KUKA KRL program: EPS_2_251825_SA30_A_20260116064111.src

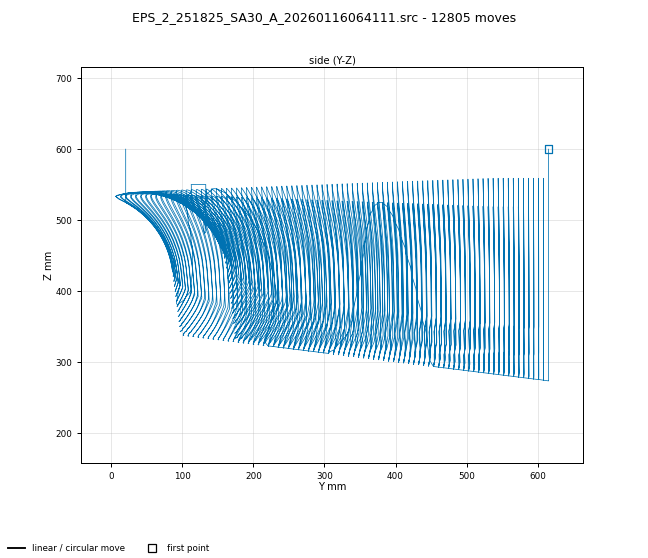
[picture p0: tool path of EPS_2_251825_SA30_A_20260116064111.src, 12805 of 12807 moves have a stored position in this frame; points joined in program order, loops and branches not executed]
&ACCESS RVP
&REL 4
&COMMENT QRS 19112012
&PARAM EDITMASK = *
DEF PART()
EXT BAS (BAS_COMMAND :IN,REAL :IN )
INT I
BAS (#INITMOV,0 )

;KUKA QRS Post kuka4.cps  Date:22-06-2017 !

File_ID=2989

QRS_PRE_INIT()

;Init var - Until changes are made in qrs_pre_init
Outlet_Square_prg=0
Inlet_1_Square_prg=0
Inlet_2_Square_prg=0
Inlet_3_Square_prg=0
Inlet_4_Square_prg=0
Inlet_5_Square_prg=0

Outlet_1={X 0.000, Y 535.490, Z 458.500, B 0.000, E1 0.000 }
Inlet_1={X 0.000, Y 538.340, Z 418.500, B 0.000, E1 194.000 }
Outlet_1_type=201
Inlet_1_type=201
;QRS#1=Sidecore dimensions
;QRS#2=200-8" PVC SDR 35
;QRS#3=200-8" PVC SDR 35
;QRS#4=
;QRS#5=
;QRS#6=
;QRS#7=
;QRS#8=
;QRS#9=12-08 PSX
;QRS#10=12-08 PSX
;QRS#11=
;QRS#12=
;QRS#13=
;QRS#14=
;QRS#15=
;QRS#16=1220x127x838 2,75'
;QRS#17=EPS Height
;QRS#18=559
;QRS#19=*
;QRS#20= UPDATED VERSION 22-06-2017
;QRS#21=*
Outlet_Square=0100
Inlet_1_Square=0100
Inlet_2_Square=0
Inlet_3_Square=0
Inlet_4_Square=0
Inlet_5_Square=0
Mill_Square=1
Outlet_Square_Prg=204
Inlet_1_Square_prg=204

QRS_INIT()

$ADVANCE=5

; T1
PTP {E1 173.624,E2 173.624}
PTP {X 0,Y 615.46,A -85,B 0,C 180,E1 173.624,E2 173.624,E3 0,E4 0,E5 0,E6 0}
QRS_SPEED_INIT()
LIN {X 0,Y 615.46,Z 600,A -85,B 0,C 180,E1 173.624,E2 173.624,E3 0,E4 0,E5 0,E6 0} C_VEL
LIN {X 0,Y 615.46,Z 283.872,A -85,B 0,C 180,E1 173.624,E2 173.624} C_VEL
LIN {X 0,Y 615.46,Z 275.69,A -85,B 0,C 180,E1 173.624,E2 173.624} C_VEL
LIN {X 0,Y 615.454,Z 273.69,A -85,B 0,C 180,E1 173.438,E2 173.438} C_VEL
LIN {X 0,Y 615.487,Z 273.682,A -85,B 0,C 180,E1 170.801,E2 170.801} C_VEL
LIN {X 0,Y 615.494,Z 273.696,A -85,B 0,C 180,E1 168.139,E2 168.139} C_VEL
LIN {X 0,Y 615.455,Z 273.694,A -85,B 0,C 180,E1 165.45,E2 165.45} C_VEL
LIN {X 0,Y 615.454,Z 273.694,A -85,B 0,C 180,E1 163.412,E2 163.412} C_VEL
LIN {X 0,Y 615.454,Z 273.694,A -85,B 0,C 180,E1 161.353,E2 161.353} C_VEL
LIN {X 0,Y 615.452,Z 273.694,A -85,B 0,C 180,E1 159.268,E2 159.268} C_VEL
LIN {X 0,Y 615.449,Z 273.694,A -85,B 0,C 180,E1 157.154,E2 157.154} C_VEL
LIN {X 0,Y 615.446,Z 273.693,A -85,B 0,C 180,E1 155.006,E2 155.006} C_VEL
LIN {X 0,Y 615.444,Z 273.692,A -85,B 0,C 180,E1 152.821,E2 152.821} C_VEL
LIN {X 0,Y 615.474,Z 273.686,A -85,B 0,C 180,E1 150.205,E2 150.205} C_VEL
LIN {X 0,Y 615.493,Z 273.698,A -85,B 0,C 180,E1 147.543,E2 147.543} C_VEL
LIN {X 0,Y 615.47,Z 273.698,A -85,B 0,C 180,E1 145.184,E2 145.184} C_VEL
LIN {X 0,Y 615.443,Z 273.695,A -85,B 0,C 180,E1 142.754,E2 142.754} C_VEL
LIN {X 0,Y 615.465,Z 273.688,A -85,B 0,C 180,E1 139.912,E2 139.912} C_VEL
LIN {X 0,Y 615.466,Z 273.699,A -85,B 0,C 180,E1 136.953,E2 136.953} C_VEL
LIN {X 0,Y 615.473,Z 273.698,A -85,B 0,C 180,E1 134.93,E2 134.93} C_VEL
LIN {X 0,Y 615.435,Z 273.695,A -85,B 0,C 180,E1 132.356,E2 132.356} C_VEL
LIN {X 0,Y 615.433,Z 273.693,A -85,B 0,C 180,E1 130.083,E2 130.083} C_VEL
LIN {X 0,Y 615.432,Z 273.693,A -85,B 0,C 180,E1 128.005,E2 128.005} C_VEL
LIN {X 0,Y 615.446,Z 273.692,A -85,B 0,C 180,E1 125.617,E2 125.617} C_VEL
LIN {X 0,Y 615.473,Z 273.691,A -85,B 0,C 180,E1 123.236,E2 123.236} C_VEL
LIN {X 0,Y 615.492,Z 273.695,A -85,B 0,C 180,E1 120.918,E2 120.918} C_VEL
LIN {X 0,Y 615.426,Z 273.696,A -85,B 0,C 180,E1 117.917,E2 117.917} C_VEL
LIN {X 0,Y 615.427,Z 273.694,A -85,B 0,C 180,E1 115.556,E2 115.556} C_VEL
LIN {X 0,Y 615.484,Z 273.692,A -85,B 0,C 180,E1 112.844,E2 112.844} C_VEL
LIN {X 0,Y 615.442,Z 273.698,A -85,B 0,C 180,E1 110.034,E2 110.034} C_VEL
LIN {X 0,Y 615.44,Z 273.698,A -85,B 0,C 180,E1 107.958,E2 107.958} C_VEL
LIN {X 0,Y 615.439,Z 273.699,A -85,B 0,C 180,E1 105.906,E2 105.906} C_VEL
LIN {X 0,Y 615.441,Z 273.699,A -85,B 0,C 180,E1 103.875,E2 103.875} C_VEL
LIN {X 0,Y 615.445,Z 273.699,A -85,B 0,C 180,E1 101.861,E2 101.861} C_VEL
LIN {X 0,Y 615.45,Z 273.699,A -85,B 0,C 180,E1 99.862,E2 99.862} C_VEL
LIN {X 0,Y 615.411,Z 273.698,A -85,B 0,C 180,E1 97.216,E2 97.216} C_VEL
LIN {X 0,Y 615.43,Z 273.697,A -85,B 0,C 180,E1 94.666,E2 94.666} C_VEL
LIN {X 0,Y 615.473,Z 275.838,A -85,B 0,C 180,E1 94.256,E2 94.256} C_VEL
LIN {X 0,Y 615.449,Z 291.323,A -85,B 0,C 180,E1 91.635,E2 91.635} C_VEL
LIN {X 0,Y 615.455,Z 306.957,A -85,B 0,C 180,E1 89.018,E2 89.018} C_VEL
LIN {X 0,Y 615.468,Z 308.181,A -85,B 0,C 180,E1 88.814,E2 88.814} C_VEL
LIN {X 0,Y 615.469,Z 414.797,A -85,B 0,C 180,E1 87.545,E2 87.545} C_VEL
LIN {X 0,Y 615.464,Z 427.886,A -85,B 0,C 180,E1 87.259,E2 87.259} C_VEL
LIN {X 0,Y 615.484,Z 440.419,A -85,B 0,C 180,E1 86.849,E2 86.849} C_VEL
LIN {X 0,Y 615.484,Z 452.453,A -85,B 0,C 180,E1 86.317,E2 86.317} C_VEL
LIN {X 0,Y 615.494,Z 463.84,A -85,B 0,C 180,E1 85.661,E2 85.661} C_VEL
LIN {X 0,Y 615.498,Z 474.118,A -85,B 0,C 180,E1 84.923,E2 84.923} C_VEL
LIN {X 0,Y 615.497,Z 481.621,A -85,B 0,C 180,E1 84.266,E2 84.266} C_VEL
LIN {X 0,Y 615.496,Z 489.878,A -85,B 0,C 180,E1 83.417,E2 83.417} C_VEL
LIN {X 0,Y 615.49,Z 497.479,A -85,B 0,C 180,E1 82.454,E2 82.454} C_VEL
LIN {X 0,Y 615.496,Z 503.742,A -85,B 0,C 180,E1 81.463,E2 81.463} C_VEL
LIN {X 0,Y 615.497,Z 508.742,A -85,B 0,C 180,E1 80.469,E2 80.469} C_VEL
LIN {X 0,Y 615.496,Z 512.615,A -85,B 0,C 180,E1 79.473,E2 79.473} C_VEL
LIN {X 0,Y 615.497,Z 514.607,A -85,B 0,C 180,E1 78.807,E2 78.807} C_VEL
LIN {X 0,Y 615.495,Z 516.186,A -85,B 0,C 180,E1 78.139,E2 78.139} C_VEL
LIN {X 0,Y 615.495,Z 517.337,A -85,B 0,C 180,E1 77.47,E2 77.47} C_VEL
LIN {X 0,Y 615.495,Z 518.354,A -85,B 0,C 180,E1 76.126,E2 76.126} C_VEL
LIN {X 0,Y 615.497,Z 518.271,A -85,B 0,C 180,E1 75.451,E2 75.451} C_VEL
LIN {X 0,Y 615.494,Z 517.731,A -85,B 0,C 180,E1 74.774,E2 74.774} C_VEL
LIN {X 0,Y 615.493,Z 515.746,A -85,B 0,C 180,E1 73.568,E2 73.568} C_VEL
LIN {X 0,Y 615.496,Z 512.453,A -85,B 0,C 180,E1 72.387,E2 72.387} C_VEL
LIN {X 0,Y 615.497,Z 508.371,A -85,B 0,C 180,E1 71.354,E2 71.354} C_VEL
LIN {X 0,Y 615.497,Z 501.94,A -85,B 0,C 180,E1 70.141,E2 70.141} C_VEL
LIN {X 0,Y 615.498,Z 494.801,A -85,B 0,C 180,E1 69.094,E2 69.094} C_VEL
LIN {X 0,Y 615.499,Z 487.402,A -85,B 0,C 180,E1 68.216,E2 68.216} C_VEL
LIN {X 0,Y 615.496,Z 477.643,A -85,B 0,C 180,E1 67.28,E2 67.28} C_VEL
LIN {X 0,Y 615.483,Z 466.81,A -85,B 0,C 180,E1 66.443,E2 66.443} C_VEL
LIN {X 0,Y 615.46,Z 456.253,A -85,B 0,C 180,E1 65.795,E2 65.795} C_VEL
LIN {X 0,Y 615.495,Z 444.674,A -85,B 0,C 180,E1 65.234,E2 65.234} C_VEL
LIN {X 0,Y 615.448,Z 431.759,A -85,B 0,C 180,E1 64.761,E2 64.761} C_VEL
LIN {X 0,Y 615.428,Z 419.153,A -85,B 0,C 180,E1 64.443,E2 64.443} C_VEL
LIN {X 0,Y 615.426,Z 403.17,A -85,B 0,C 180,E1 64.213,E2 64.213} C_VEL
LIN {X 0,Y 615.497,Z 308.127,A -85,B 0,C 180,E1 63.089,E2 63.089} C_VEL
LIN {X 0,Y 615.459,Z 292.076,A -85,B 0,C 180,E1 60.401,E2 60.401} C_VEL
LIN {X 0,Y 615.486,Z 275.929,A -85,B 0,C 180,E1 57.67,E2 57.67} C_VEL
LIN {X 0,Y 615.48,Z 273.686,A -85,B 0,C 180,E1 57.251,E2 57.251} C_VEL
LIN {X 0,Y 615.479,Z 273.686,A -85,B 0,C 180,E1 55.184,E2 55.184} C_VEL
LIN {X 0,Y 615.489,Z 273.68,A -85,B 0,C 180,E1 52.758,E2 52.758} C_VEL
LIN {X 0,Y 615.477,Z 273.694,A -85,B 0,C 180,E1 49.913,E2 49.913} C_VEL
LIN {X 0,Y 615.49,Z 273.698,A -85,B 0,C 180,E1 47.647,E2 47.647} C_VEL
LIN {X 0,Y 615.477,Z 273.688,A -85,B 0,C 180,E1 44.931,E2 44.931} C_VEL
LIN {X 0,Y 615.477,Z 273.685,A -85,B 0,C 180,E1 42.079,E2 42.079} C_VEL
LIN {X 0,Y 615.474,Z 273.69,A -85,B 0,C 180,E1 39.751,E2 39.751} C_VEL
LIN {X 0,Y 615.481,Z 273.694,A -85,B 0,C 180,E1 36.936,E2 36.936} C_VEL
LIN {X 0,Y 615.49,Z 273.68,A -85,B 0,C 180,E1 34.022,E2 34.022} C_VEL
LIN {X 0,Y 615.481,Z 273.702,A -85,B 0,C 180,E1 31.085,E2 31.085} C_VEL
LIN {X 0,Y 615.476,Z 273.689,A -85,B 0,C 180,E1 28.449,E2 28.449} C_VEL
LIN {X 0,Y 615.488,Z 273.681,A -85,B 0,C 180,E1 25.716,E2 25.716} C_VEL
LIN {X 0,Y 615.491,Z 273.699,A -85,B 0,C 180,E1 22.845,E2 22.845} C_VEL
LIN {X 0,Y 615.477,Z 273.686,A -85,B 0,C 180,E1 20.033,E2 20.033} C_VEL
LIN {X 0,Y 615.477,Z 273.685,A -85,B 0,C 180,E1 17.271,E2 17.271} C_VEL
LIN {X 0,Y 615.491,Z 273.7,A -85,B 0,C 180,E1 14.549,E2 14.549} C_VEL
LIN {X 0,Y 615.474,Z 273.688,A -85,B 0,C 180,E1 11.861,E2 11.861} C_VEL
LIN {X 0,Y 615.491,Z 273.68,A -85,B 0,C 180,E1 9.199,E2 9.199} C_VEL
LIN {X 0,Y 615.476,Z 273.694,A -85,B 0,C 180,E1 6.557,E2 6.557} C_VEL
LIN {X 0,Y 615.482,Z 273.695,A -85,B 0,C 180,E1 3.929,E2 3.929} C_VEL
LIN {X 0,Y 615.48,Z 273.683,A -85,B 0,C 180,E1 1.309,E2 1.309} C_VEL
LIN {X 0,Y 615.482,Z 273.684,A -85,B 0,C 180,E1 -1.309,E2 -1.309} C_VEL
LIN {X 0,Y 615.487,Z 273.696,A -85,B 0,C 180,E1 -3.928,E2 -3.928} C_VEL
LIN {X 0,Y 615.475,Z 273.692,A -85,B 0,C 180,E1 -6.57,E2 -6.57} C_VEL
LIN {X 0,Y 615.49,Z 273.68,A -85,B 0,C 180,E1 -9.199,E2 -9.199} C_VEL
LIN {X 0,Y 615.477,Z 273.689,A -85,B 0,C 180,E1 -11.861,E2 -11.861} C_VEL
LIN {X 0,Y 615.489,Z 273.698,A -85,B 0,C 180,E1 -14.549,E2 -14.549} C_VEL
LIN {X 0,Y 615.475,Z 273.685,A -85,B 0,C 180,E1 -17.271,E2 -17.271} C_VEL
LIN {X 0,Y 615.479,Z 273.686,A -85,B 0,C 180,E1 -20.033,E2 -20.033} C_VEL
LIN {X 0,Y 615.486,Z 273.697,A -85,B 0,C 180,E1 -22.845,E2 -22.845} C_VEL
LIN {X 0,Y 615.487,Z 273.681,A -85,B 0,C 180,E1 -25.716,E2 -25.716} C_VEL
LIN {X 0,Y 615.485,Z 273.695,A -85,B 0,C 180,E1 -28.658,E2 -28.658} C_VEL
LIN {X 0,Y 615.481,Z 273.699,A -85,B 0,C 180,E1 -31.085,E2 -31.085} C_VEL
LIN {X 0,Y 615.489,Z 273.68,A -85,B 0,C 180,E1 -34.022,E2 -34.022} C_VEL
LIN {X 0,Y 615.484,Z 273.695,A -85,B 0,C 180,E1 -36.936,E2 -36.936} C_VEL
LIN {X 0,Y 615.47,Z 273.689,A -85,B 0,C 180,E1 -39.752,E2 -39.752} C_VEL
LIN {X 0,Y 615.493,Z 273.679,A -85,B 0,C 180,E1 -42.353,E2 -42.353} C_VEL
LIN {X 0,Y 615.481,Z 273.692,A -85,B 0,C 180,E1 -45.069,E2 -45.069} C_VEL
LIN {X 0,Y 615.47,Z 273.692,A -85,B 0,C 180,E1 -47.922,E2 -47.922} C_VEL
LIN {X 0,Y 615.471,Z 273.686,A -85,B 0,C 180,E1 -50.249,E2 -50.249} C_VEL
LIN {X 0,Y 615.481,Z 273.686,A -85,B 0,C 180,E1 -53.065,E2 -53.065} C_VEL
LIN {X 0,Y 615.48,Z 273.696,A -85,B 0,C 180,E1 -55.978,E2 -55.978} C_VEL
LIN {X 0,Y 615.469,Z 273.69,A -85,B 0,C 180,E1 -58.313,E2 -58.313} C_VEL
LIN {X 0,Y 615.47,Z 273.686,A -85,B 0,C 180,E1 -60.593,E2 -60.593} C_VEL
LIN {X 0,Y 615.486,Z 273.681,A -85,B 0,C 180,E1 -62.956,E2 -62.956} C_VEL
LIN {X 0,Y 615.481,Z 273.692,A -85,B 0,C 180,E1 -65.728,E2 -65.728} C_VEL
LIN {X 0,Y 615.487,Z 273.753,A -85,B 0,C 180,E1 -67.437,E2 -67.437} C_VEL
LIN {X 0,Y 615.455,Z 293.69,A -85,B 0,C 180,E1 -70.14,E2 -70.14} C_VEL
LIN {X 0,Y 615.472,Z 313.075,A -85,B 0,C 180,E1 -72.729,E2 -72.729} C_VEL
LIN {X 0,Y 615.493,Z 334.915,A -85,B 0,C 180,E1 -75.606,E2 -75.606} C_VEL
LIN {X 0,Y 615.471,Z 346.466,A -85,B 0,C 180,E1 -77.113,E2 -77.113} C_VEL
LIN {X 0,Y 615.457,Z 454.819,A -85,B 0,C 180,E1 -78.41,E2 -78.41} C_VEL
LIN {X 0,Y 615.456,Z 467.337,A -85,B 0,C 180,E1 -78.681,E2 -78.681} C_VEL
LIN {X 0,Y 615.483,Z 480.687,A -85,B 0,C 180,E1 -79.115,E2 -79.115} C_VEL
LIN {X 0,Y 615.492,Z 492.47,A -85,B 0,C 180,E1 -79.639,E2 -79.639} C_VEL
LIN {X 0,Y 615.483,Z 503.99,A -85,B 0,C 180,E1 -80.303,E2 -80.303} C_VEL
LIN {X 0,Y 615.499,Z 514.336,A -85,B 0,C 180,E1 -81.049,E2 -81.049} C_VEL
LIN {X 0,Y 615.497,Z 522.688,A -85,B 0,C 180,E1 -81.794,E2 -81.794} C_VEL
LIN {X 0,Y 615.498,Z 530.603,A -85,B 0,C 180,E1 -82.619,E2 -82.619} C_VEL
LIN {X 0,Y 615.491,Z 538.201,A -85,B 0,C 180,E1 -83.608,E2 -83.608} C_VEL
LIN {X 0,Y 615.498,Z 545.202,A -85,B 0,C 180,E1 -84.758,E2 -84.758} C_VEL
LIN {X 0,Y 615.493,Z 549.85,A -85,B 0,C 180,E1 -85.743,E2 -85.743} C_VEL
LIN {X 0,Y 615.494,Z 553.397,A -85,B 0,C 180,E1 -86.727,E2 -86.727} C_VEL
LIN {X 0,Y 615.497,Z 555.232,A -85,B 0,C 180,E1 -87.382,E2 -87.382} C_VEL
LIN {X 0,Y 615.497,Z 556.607,A -85,B 0,C 180,E1 -88.036,E2 -88.036} C_VEL
LIN {X 0,Y 615.496,Z 558.173,A -85,B 0,C 180,E1 -89.345,E2 -89.345} C_VEL
LIN {X 0,Y 615.494,Z 558.389,A -85,B 0,C 180,E1 -90,E2 -90} C_VEL
LIN {X 0,Y 615.495,Z 557.581,A -85,B 0,C 180,E1 -91.308,E2 -91.308} C_VEL
LIN {X 0,Y 615.497,Z 556.609,A -85,B 0,C 180,E1 -91.963,E2 -91.963} C_VEL
LIN {X 0,Y 615.497,Z 555.234,A -85,B 0,C 180,E1 -92.617,E2 -92.617} C_VEL
LIN {X 0,Y 615.496,Z 552.351,A -85,B 0,C 180,E1 -93.6,E2 -93.6} C_VEL
LIN {X 0,Y 615.498,Z 548.444,A -85,B 0,C 180,E1 -94.584,E2 -94.584} C_VEL
LIN {X 0,Y 615.499,Z 543.408,A -85,B 0,C 180,E1 -95.569,E2 -95.569} C_VEL
LIN {X 0,Y 615.49,Z 536.913,A -85,B 0,C 180,E1 -96.578,E2 -96.578} C_VEL
LIN {X 0,Y 615.497,Z 529.138,A -85,B 0,C 180,E1 -97.545,E2 -97.545} C_VEL
LIN {X 0,Y 615.498,Z 519.264,A -85,B 0,C 180,E1 -98.536,E2 -98.536} C_VEL
LIN {X 0,Y 615.495,Z 508.874,A -85,B 0,C 180,E1 -99.364,E2 -99.364} C_VEL
LIN {X 0,Y 615.482,Z 498.586,A -85,B 0,C 180,E1 -100.028,E2 -100.028} C_VEL
LIN {X 0,Y 615.495,Z 487.147,A -85,B 0,C 180,E1 -100.616,E2 -100.616} C_VEL
LIN {X 0,Y 615.467,Z 475.37,A -85,B 0,C 180,E1 -101.077,E2 -101.077} C_VEL
LIN {X 0,Y 615.455,Z 462.275,A -85,B 0,C 180,E1 -101.443,E2 -101.443} C_VEL
LIN {X 0,Y 615.461,Z 449,A -85,B 0,C 180,E1 -101.673,E2 -101.673} C_VEL
LIN {X 0,Y 615.471,Z 346.473,A -85,B 0,C 180,E1 -102.886,E2 -102.886} C_VEL
LIN {X 0,Y 615.455,Z 325.995,A -85,B 0,C 180,E1 -105.565,E2 -105.565} C_VEL
LIN {X 0,Y 615.481,Z 305.477,A -85,B 0,C 180,E1 -108.281,E2 -108.281} C_VEL
LIN {X 0,Y 615.468,Z 283.349,A -85,B 0,C 180,E1 -111.256,E2 -111.256} C_VEL
LIN {X 0,Y 615.489,Z 273.682,A -85,B 0,C 180,E1 -112.593,E2 -112.593} C_VEL
LIN {X 0,Y 615.485,Z 273.681,A -85,B 0,C 180,E1 -114.991,E2 -114.991} C_VEL
LIN {X 0,Y 615.482,Z 273.7,A -85,B 0,C 180,E1 -117.914,E2 -117.914} C_VEL
LIN {X 0,Y 615.493,Z 273.699,A -85,B 0,C 180,E1 -120.159,E2 -120.159} C_VEL
LIN {X 0,Y 615.481,Z 273.693,A -85,B 0,C 180,E1 -122.457,E2 -122.457} C_VEL
LIN {X 0,Y 615.479,Z 273.686,A -85,B 0,C 180,E1 -124.814,E2 -124.814} C_VEL
LIN {X 0,Y 615.49,Z 273.68,A -85,B 0,C 180,E1 -127.241,E2 -127.241} C_VEL
LIN {X 0,Y 615.478,Z 273.695,A -85,B 0,C 180,E1 -130.088,E2 -130.088} C_VEL
LIN {X 0,Y 615.494,Z 273.699,A -85,B 0,C 180,E1 -132.351,E2 -132.351} C_VEL
LIN {X 0,Y 615.475,Z 273.687,A -85,B 0,C 180,E1 -135.068,E2 -135.068} C_VEL
LIN {X 0,Y 615.48,Z 273.685,A -85,B 0,C 180,E1 -137.919,E2 -137.919} C_VEL
LIN {X 0,Y 615.476,Z 273.692,A -85,B 0,C 180,E1 -140.249,E2 -140.249} C_VEL
LIN {X 0,Y 615.474,Z 273.693,A -85,B 0,C 180,E1 -143.063,E2 -143.063} C_VEL
LIN {X 0,Y 615.491,Z 273.681,A -85,B 0,C 180,E1 -145.978,E2 -145.978} C_VEL
LIN {X 0,Y 615.486,Z 273.701,A -85,B 0,C 180,E1 -148.912,E2 -148.912} C_VEL
LIN {X 0,Y 615.467,Z 273.688,A -85,B 0,C 180,E1 -151.551,E2 -151.551} C_VEL
LIN {X 0,Y 615.49,Z 273.682,A -85,B 0,C 180,E1 -154.284,E2 -154.284} C_VEL
LIN {X 0,Y 615.483,Z 273.7,A -85,B 0,C 180,E1 -157.155,E2 -157.155} C_VEL
LIN {X 0,Y 615.47,Z 273.685,A -85,B 0,C 180,E1 -159.967,E2 -159.967} C_VEL
LIN {X 0,Y 615.484,Z 273.687,A -85,B 0,C 180,E1 -162.729,E2 -162.729} C_VEL
LIN {X 0,Y 615.48,Z 273.698,A -85,B 0,C 180,E1 -165.451,E2 -165.451} C_VEL
LIN {X 0,Y 615.464,Z 273.687,A -85,B 0,C 180,E1 -168.139,E2 -168.139} C_VEL
LIN {X 0,Y 615.493,Z 273.682,A -85,B 0,C 180,E1 -170.801,E2 -170.801} C_VEL
LIN {X 0,Y 615.496,Z 273.699,A -85,B 0,C 180,E1 -173.443,E2 -173.443} C_VEL
LIN {X 0,Y 615.461,Z 273.692,A -85,B 0,C 180,E1 -176.071,E2 -176.071} C_VEL
LIN {X 0,Y 615.473,Z 273.684,A -85,B 0,C 180,E1 -178.691,E2 -178.691} C_VEL
LIN {X 0,Y 615.489,Z 273.688,A -85,B 0,C 180,E1 -181.309,E2 -181.309} C_VEL
LIN {X 0,Y 615.481,Z 273.698,A -85,B 0,C 180,E1 -183.929,E2 -183.929} C_VEL
LIN {X 0,Y 615.454,Z 273.69,A -85,B 0,C 180,E1 -186.562,E2 -186.562} C_VEL
LIN {X 0,Y 614.798,Z 273.834,A -85,B 0,C 180,E1 -187.108,E2 -187.108} C_VEL
LIN {X 0,Y 611.98,Z 274.257,A -85,B 0,C 180,E1 -187.994,E2 -187.994} C_VEL
LIN {X 0,Y 609.589,Z 274.561,A -85,B 0,C 180,E1 -188.707,E2 -188.707} C_VEL
LIN {X 0,Y 608.551,Z 274.677,A -85,B 0,C 180,E1 -189.256,E2 -189.256} C_VEL
LIN {X 0,Y 608.461,Z 274.688,A -85,B 0,C 180,E1 -189.442,E2 -189.442} C_VEL
LIN {X 0,Y 608.459,Z 274.698,A -85,B 0,C 180,E1 -192,E2 -192} C_VEL
LIN {X 0,Y 608.422,Z 274.692,A -85,B 0,C 180,E1 -194.722,E2 -194.722} C_VEL
LIN {X 0,Y 608.421,Z 274.692,A -85,B 0,C 180,E1 -196.785,E2 -196.785} C_VEL
LIN {X 0,Y 608.441,Z 274.689,A -85,B 0,C 180,E1 -199.571,E2 -199.571} C_VEL
LIN {X 0,Y 608.449,Z 274.695,A -85,B 0,C 180,E1 -202.477,E2 -202.477} C_VEL
LIN {X 0,Y 608.439,Z 274.695,A -85,B 0,C 180,E1 -204.572,E2 -204.572} C_VEL
LIN {X 0,Y 608.423,Z 274.691,A -85,B 0,C 180,E1 -207.2,E2 -207.2} C_VEL
LIN {X 0,Y 608.459,Z 274.687,A -85,B 0,C 180,E1 -209.78,E2 -209.78} C_VEL
LIN {X 0,Y 608.464,Z 274.697,A -85,B 0,C 180,E1 -212.525,E2 -212.525} C_VEL
LIN {X 0,Y 608.414,Z 274.692,A -85,B 0,C 180,E1 -215.28,E2 -215.28} C_VEL
LIN {X 0,Y 608.445,Z 274.687,A -85,B 0,C 180,E1 -217.748,E2 -217.748} C_VEL
LIN {X 0,Y 608.442,Z 274.692,A -85,B 0,C 180,E1 -220.33,E2 -220.33} C_VEL
LIN {X 0,Y 608.435,Z 274.697,A -85,B 0,C 180,E1 -222.962,E2 -222.962} C_VEL
LIN {X 0,Y 608.414,Z 274.691,A -85,B 0,C 180,E1 -225.741,E2 -225.741} C_VEL
LIN {X 0,Y 608.418,Z 274.691,A -85,B 0,C 180,E1 -227.936,E2 -227.936} C_VEL
LIN {X 0,Y 608.44,Z 274.694,A -85,B 0,C 180,E1 -230.706,E2 -230.706} C_VEL
LIN {X 0,Y 608.454,Z 274.698,A -85,B 0,C 180,E1 -233.086,E2 -233.086} C_VEL
LIN {X 0,Y 608.448,Z 274.692,A -85,B 0,C 180,E1 -235.53,E2 -235.53} C_VEL
LIN {X 0,Y 608.424,Z 274.691,A -85,B 0,C 180,E1 -237.904,E2 -237.904} C_VEL
LIN {X 0,Y 608.414,Z 274.691,A -85,B 0,C 180,E1 -240.219,E2 -240.219} C_VEL
LIN {X 0,Y 608.441,Z 274.69,A -85,B 0,C 180,E1 -242.8,E2 -242.8} C_VEL
LIN {X 0,Y 608.439,Z 274.692,A -85,B 0,C 180,E1 -245.856,E2 -245.856} C_VEL
LIN {X 0,Y 608.42,Z 274.691,A -85,B 0,C 180,E1 -248.307,E2 -248.307} C_VEL
LIN {X 0,Y 608.402,Z 274.693,A -85,B 0,C 180,E1 -250.429,E2 -250.429} C_VEL
LIN {X 0,Y 608.401,Z 274.693,A -85,B 0,C 180,E1 -252.523,E2 -252.523} C_VEL
LIN {X 0,Y 608.415,Z 274.691,A -85,B 0,C 180,E1 -254.593,E2 -254.593} C_VEL
LIN {X 0,Y 608.453,Z 274.69,A -85,B 0,C 180,E1 -257.323,E2 -257.323} C_VEL
LIN {X 0,Y 608.426,Z 274.697,A -85,B 0,C 180,E1 -260.023,E2 -260.023} C_VEL
LIN {X 0,Y 608.398,Z 274.694,A -85,B 0,C 180,E1 -262.7,E2 -262.7} C_VEL
LIN {X 0,Y 608.406,Z 274.734,A -85,B 0,C 180,E1 -265.321,E2 -265.321} C_VEL
LIN {X 0,Y 608.463,Z 290.468,A -85,B 0,C 180,E1 -268.015,E2 -268.015} C_VEL
LIN {X 0,Y 608.428,Z 306.156,A -85,B 0,C 180,E1 -270.662,E2 -270.662} C_VEL
LIN {X 0,Y 608.44,Z 308.374,A -85,B 0,C 180,E1 -271.035,E2 -271.035} C_VEL
LIN {X 0,Y 608.517,Z 414.73,A -85,B 0,C 180,E1 -272.317,E2 -272.317} C_VEL
LIN {X 0,Y 608.499,Z 427.883,A -85,B 0,C 180,E1 -272.607,E2 -272.607} C_VEL
LIN {X 0,Y 608.522,Z 440.458,A -85,B 0,C 180,E1 -273.021,E2 -273.021} C_VEL
LIN {X 0,Y 608.501,Z 452.549,A -85,B 0,C 180,E1 -273.56,E2 -273.56} C_VEL
LIN {X 0,Y 608.505,Z 463.991,A -85,B 0,C 180,E1 -274.223,E2 -274.223} C_VEL
LIN {X 0,Y 608.476,Z 474.332,A -85,B 0,C 180,E1 -274.97,E2 -274.97} C_VEL
LIN {X 0,Y 608.47,Z 481.894,A -85,B 0,C 180,E1 -275.635,E2 -275.635} C_VEL
LIN {X 0,Y 608.468,Z 490.286,A -85,B 0,C 180,E1 -276.503,E2 -276.503} C_VEL
LIN {X 0,Y 608.445,Z 497.863,A -85,B 0,C 180,E1 -277.467,E2 -277.467} C_VEL
LIN {X 0,Y 608.456,Z 503.226,A -85,B 0,C 180,E1 -278.302,E2 -278.302} C_VEL
LIN {X 0,Y 608.432,Z 508.491,A -85,B 0,C 180,E1 -279.307,E2 -279.307} C_VEL
LIN {X 0,Y 608.438,Z 512.582,A -85,B 0,C 180,E1 -280.314,E2 -280.314} C_VEL
LIN {X 0,Y 608.426,Z 515.619,A -85,B 0,C 180,E1 -281.325,E2 -281.325} C_VEL
LIN {X 0,Y 608.44,Z 517.104,A -85,B 0,C 180,E1 -282.001,E2 -282.001} C_VEL
LIN {X 0,Y 608.44,Z 518.765,A -85,B 0,C 180,E1 -283.357,E2 -283.357} C_VEL
LIN {X 0,Y 608.426,Z 519,A -85,B 0,C 180,E1 -284.039,E2 -284.039} C_VEL
LIN {X 0,Y 608.418,Z 518.773,A -85,B 0,C 180,E1 -284.722,E2 -284.722} C_VEL
LIN {X 0,Y 608.417,Z 518.138,A -85,B 0,C 180,E1 -285.408,E2 -285.408} C_VEL
LIN {X 0,Y 608.422,Z 516.213,A -85,B 0,C 180,E1 -286.513,E2 -286.513} C_VEL
LIN {X 0,Y 608.428,Z 512.4,A -85,B 0,C 180,E1 -287.825,E2 -287.825} C_VEL
LIN {X 0,Y 608.434,Z 508.066,A -85,B 0,C 180,E1 -288.871,E2 -288.871} C_VEL
LIN {X 0,Y 608.437,Z 502.408,A -85,B 0,C 180,E1 -289.923,E2 -289.923} C_VEL
LIN {X 0,Y 608.452,Z 495.215,A -85,B 0,C 180,E1 -290.982,E2 -290.982} C_VEL
LIN {X 0,Y 608.455,Z 487.764,A -85,B 0,C 180,E1 -291.87,E2 -291.87} C_VEL
LIN {X 0,Y 608.472,Z 477.846,A -85,B 0,C 180,E1 -292.827,E2 -292.827} C_VEL
LIN {X 0,Y 608.483,Z 467.072,A -85,B 0,C 180,E1 -293.664,E2 -293.664} C_VEL
LIN {X 0,Y 608.488,Z 455.363,A -85,B 0,C 180,E1 -294.38,E2 -294.38} C_VEL
LIN {X 0,Y 608.525,Z 442.767,A -85,B 0,C 180,E1 -294.978,E2 -294.978} C_VEL
LIN {X 0,Y 608.491,Z 430.021,A -85,B 0,C 180,E1 -295.424,E2 -295.424} C_VEL
LIN {X 0,Y 608.492,Z 417.05,A -85,B 0,C 180,E1 -295.731,E2 -295.731} C_VEL
LIN {X 0,Y 608.491,Z 394.967,A -85,B 0,C 180,E1 -296.021,E2 -296.021} C_VEL
LIN {X 0,Y 608.508,Z 308.74,A -85,B 0,C 180,E1 -297.042,E2 -297.042} C_VEL
LIN {X 0,Y 608.46,Z 308.242,A -85,B 0,C 180,E1 -297.077,E2 -297.077} C_VEL
LIN {X 0,Y 608.456,Z 293.33,A -85,B 0,C 180,E1 -299.59,E2 -299.59} C_VEL
LIN {X 0,Y 608.486,Z 277.391,A -85,B 0,C 180,E1 -302.309,E2 -302.309} C_VEL
LIN {X 0,Y 608.454,Z 274.688,A -85,B 0,C 180,E1 -302.801,E2 -302.801} C_VEL
LIN {X 0,Y 608.433,Z 274.689,A -85,B 0,C 180,E1 -305.278,E2 -305.278} C_VEL
LIN {X 0,Y 608.466,Z 274.687,A -85,B 0,C 180,E1 -307.747,E2 -307.747} C_VEL
LIN {X 0,Y 608.446,Z 274.698,A -85,B 0,C 180,E1 -310.328,E2 -310.328} C_VEL
LIN {X 0,Y 608.473,Z 274.684,A -85,B 0,C 180,E1 -313.309,E2 -313.309} C_VEL
LIN {X 0,Y 608.461,Z 274.689,A -85,B 0,C 180,E1 -316.13,E2 -316.13} C_VEL
LIN {X 0,Y 608.452,Z 274.695,A -85,B 0,C 180,E1 -318.823,E2 -318.823} C_VEL
LIN {X 0,Y 608.465,Z 274.685,A -85,B 0,C 180,E1 -321.76,E2 -321.76} C_VEL
LIN {X 0,Y 608.445,Z 274.687,A -85,B 0,C 180,E1 -323.955,E2 -323.955} C_VEL
LIN {X 0,Y 608.446,Z 274.689,A -85,B 0,C 180,E1 -326.328,E2 -326.328} C_VEL
LIN {X 0,Y 608.445,Z 274.694,A -85,B 0,C 180,E1 -328.732,E2 -328.732} C_VEL
LIN {X 0,Y 608.467,Z 274.69,A -85,B 0,C 180,E1 -331.381,E2 -331.381} C_VEL
LIN {X 0,Y 608.442,Z 274.688,A -85,B 0,C 180,E1 -333.964,E2 -333.964} C_VEL
LIN {X 0,Y 608.462,Z 274.685,A -85,B 0,C 180,E1 -336.155,E2 -336.155} C_VEL
LIN {X 0,Y 608.455,Z 274.692,A -85,B 0,C 180,E1 -339.018,E2 -339.018} C_VEL
LIN {X 0,Y 608.445,Z 274.691,A -85,B 0,C 180,E1 -341.828,E2 -341.828} C_VEL
LIN {X 0,Y 608.464,Z 274.685,A -85,B 0,C 180,E1 -344.594,E2 -344.594} C_VEL
LIN {X 0,Y 608.473,Z 274.691,A -85,B 0,C 180,E1 -347.323,E2 -347.323} C_VEL
LIN {X 0,Y 608.447,Z 274.692,A -85,B 0,C 180,E1 -350.022,E2 -350.022} C_VEL
LIN {X 0,Y 608.462,Z 274.685,A -85,B 0,C 180,E1 -352.701,E2 -352.701} C_VEL
LIN {X 0,Y 608.447,Z 274.69,A -85,B 0,C 180,E1 -355.362,E2 -355.362} C_VEL
LIN {X 0,Y 608.458,Z 274.695,A -85,B 0,C 180,E1 -358.014,E2 -358.014} C_VEL
LIN {X 0,Y 608.469,Z 274.685,A -85,B 0,C 180,E1 -360.662,E2 -360.662} C_VEL
LIN {X 0,Y 608.48,Z 274.683,A -85,B 0,C 180,E1 -363.311,E2 -363.311} C_VEL
LIN {X 0,Y 608.452,Z 274.694,A -85,B 0,C 180,E1 -365.967,E2 -365.967} C_VEL
LIN {X 0,Y 608.451,Z 274.691,A -85,B 0,C 180,E1 -368.636,E2 -368.636} C_VEL
LIN {X 0,Y 608.474,Z 274.683,A -85,B 0,C 180,E1 -371.324,E2 -371.324} C_VEL
LIN {X 0,Y 608.467,Z 274.689,A -85,B 0,C 180,E1 -374.038,E2 -374.038} C_VEL
LIN {X 0,Y 608.472,Z 274.69,A -85,B 0,C 180,E1 -376.784,E2 -376.784} C_VEL
LIN {X 0,Y 608.444,Z 274.687,A -85,B 0,C 180,E1 -379.571,E2 -379.571} C_VEL
LIN {X 0,Y 608.476,Z 274.69,A -85,B 0,C 180,E1 -382.405,E2 -382.405} C_VEL
LIN {X 0,Y 608.448,Z 274.695,A -85,B 0,C 180,E1 -384.571,E2 -384.571} C_VEL
LIN {X 0,Y 608.472,Z 274.689,A -85,B 0,C 180,E1 -387.206,E2 -387.206} C_VEL
LIN {X 0,Y 608.466,Z 274.684,A -85,B 0,C 180,E1 -389.972,E2 -389.972} C_VEL
LIN {X 0,Y 608.451,Z 274.696,A -85,B 0,C 180,E1 -392.88,E2 -392.88} C_VEL
LIN {X 0,Y 608.433,Z 274.697,A -85,B 0,C 180,E1 -395.278,E2 -395.278} C_VEL
LIN {X 0,Y 608.467,Z 274.687,A -85,B 0,C 180,E1 -397.747,E2 -397.747} C_VEL
LIN {X 0,Y 608.446,Z 274.687,A -85,B 0,C 180,E1 -400.328,E2 -400.328} C_VEL
LIN {X 0,Y 608.478,Z 274.695,A -85,B 0,C 180,E1 -403.31,E2 -403.31} C_VEL
LIN {X 0,Y 608.458,Z 274.687,A -85,B 0,C 180,E1 -406.13,E2 -406.13} C_VEL
LIN {X 0,Y 608.455,Z 274.687,A -85,B 0,C 180,E1 -408.823,E2 -408.823} C_VEL
LIN {X 0,Y 608.459,Z 274.694,A -85,B 0,C 180,E1 -411.761,E2 -411.761} C_VEL
LIN {X 0,Y 608.444,Z 274.694,A -85,B 0,C 180,E1 -413.955,E2 -413.955} C_VEL
LIN {X 0,Y 608.445,Z 274.689,A -85,B 0,C 180,E1 -416.328,E2 -416.328} C_VEL
LIN {X 0,Y 608.446,Z 274.687,A -85,B 0,C 180,E1 -418.733,E2 -418.733} C_VEL
LIN {X 0,Y 608.471,Z 274.687,A -85,B 0,C 180,E1 -421.381,E2 -421.381} C_VEL
LIN {X 0,Y 608.438,Z 274.7,A -85,B 0,C 180,E1 -423.964,E2 -423.964} C_VEL
LIN {X 0,Y 608.464,Z 274.696,A -85,B 0,C 180,E1 -426.155,E2 -426.155} C_VEL
LIN {X 0,Y 608.507,Z 274.819,A -85,B 0,C 180,E1 -427.312,E2 -427.312} C_VEL
LIN {X 0,Y 608.524,Z 292.405,A -85,B 0,C 180,E1 -429.728,E2 -429.728} C_VEL
LIN {X 0,Y 608.51,Z 311.822,A -85,B 0,C 180,E1 -432.351,E2 -432.351} C_VEL
LIN {X 0,Y 608.496,Z 332.533,A -85,B 0,C 180,E1 -435.109,E2 -435.109} C_VEL
LIN {X 0,Y 608.454,Z 346.61,A -85,B 0,C 180,E1 -436.962,E2 -436.962} C_VEL
LIN {X 0,Y 608.566,Z 386.466,A -85,B 0,C 180,E1 -437.452,E2 -437.452} C_VEL
LIN {X 0,Y 608.522,Z 454.929,A -85,B 0,C 180,E1 -438.276,E2 -438.276} C_VEL
LIN {X 0,Y 608.491,Z 468.204,A -85,B 0,C 180,E1 -438.571,E2 -438.571} C_VEL
LIN {X 0,Y 608.511,Z 480.649,A -85,B 0,C 180,E1 -438.983,E2 -438.983} C_VEL
LIN {X 0,Y 608.514,Z 492.628,A -85,B 0,C 180,E1 -439.519,E2 -439.519} C_VEL
LIN {X 0,Y 608.471,Z 504.192,A -85,B 0,C 180,E1 -440.191,E2 -440.191} C_VEL
LIN {X 0,Y 608.485,Z 514.589,A -85,B 0,C 180,E1 -440.945,E2 -440.945} C_VEL
LIN {X 0,Y 608.459,Z 522.998,A -85,B 0,C 180,E1 -441.698,E2 -441.698} C_VEL
LIN {X 0,Y 608.471,Z 530.957,A -85,B 0,C 180,E1 -442.533,E2 -442.533} C_VEL
LIN {X 0,Y 608.437,Z 538.297,A -85,B 0,C 180,E1 -443.486,E2 -443.486} C_VEL
LIN {X 0,Y 608.45,Z 543.864,A -85,B 0,C 180,E1 -444.365,E2 -444.365} C_VEL
LIN {X 0,Y 608.432,Z 548.948,A -85,B 0,C 180,E1 -445.362,E2 -445.362} C_VEL
LIN {X 0,Y 608.449,Z 552.895,A -85,B 0,C 180,E1 -446.357,E2 -446.357} C_VEL
LIN {X 0,Y 608.425,Z 555.808,A -85,B 0,C 180,E1 -447.351,E2 -447.351} C_VEL
LIN {X 0,Y 608.442,Z 557.201,A -85,B 0,C 180,E1 -448.014,E2 -448.014} C_VEL
LIN {X 0,Y 608.438,Z 558.783,A -85,B 0,C 180,E1 -449.338,E2 -449.338} C_VEL
LIN {X 0,Y 608.434,Z 559,A -85,B 0,C 180,E1 -450,E2 -450} C_VEL
LIN {X 0,Y 608.448,Z 558.184,A -85,B 0,C 180,E1 -451.323,E2 -451.323} C_VEL
LIN {X 0,Y 608.442,Z 557.202,A -85,B 0,C 180,E1 -451.985,E2 -451.985} C_VEL
LIN {X 0,Y 608.425,Z 555.81,A -85,B 0,C 180,E1 -452.648,E2 -452.648} C_VEL
LIN {X 0,Y 608.449,Z 552.898,A -85,B 0,C 180,E1 -453.642,E2 -453.642} C_VEL
LIN {X 0,Y 608.432,Z 548.952,A -85,B 0,C 180,E1 -454.637,E2 -454.637} C_VEL
LIN {X 0,Y 608.437,Z 542.88,A -85,B 0,C 180,E1 -455.8,E2 -455.8} C_VEL
LIN {X 0,Y 608.46,Z 536.239,A -85,B 0,C 180,E1 -456.799,E2 -456.799} C_VEL
LIN {X 0,Y 608.455,Z 527.994,A -85,B 0,C 180,E1 -457.8,E2 -457.8} C_VEL
LIN {X 0,Y 608.477,Z 517.605,A -85,B 0,C 180,E1 -458.803,E2 -458.803} C_VEL
LIN {X 0,Y 608.488,Z 506.756,A -85,B 0,C 180,E1 -459.64,E2 -459.64} C_VEL
LIN {X 0,Y 608.491,Z 495.785,A -85,B 0,C 180,E1 -460.312,E2 -460.312} C_VEL
LIN {X 0,Y 608.534,Z 483.808,A -85,B 0,C 180,E1 -460.888,E2 -460.888} C_VEL
LIN {X 0,Y 608.505,Z 471.899,A -85,B 0,C 180,E1 -461.323,E2 -461.323} C_VEL
LIN {X 0,Y 608.507,Z 459.546,A -85,B 0,C 180,E1 -461.639,E2 -461.639} C_VEL
LIN {X 0,Y 608.531,Z 443.787,A -85,B 0,C 180,E1 -461.871,E2 -461.871} C_VEL
LIN {X 0,Y 608.508,Z 347.199,A -85,B 0,C 180,E1 -463.015,E2 -463.015} C_VEL
LIN {X 0,Y 608.454,Z 346.133,A -85,B 0,C 180,E1 -463.101,E2 -463.101} C_VEL
LIN {X 0,Y 608.467,Z 327.363,A -85,B 0,C 180,E1 -465.577,E2 -465.577} C_VEL
LIN {X 0,Y 608.508,Z 307.946,A -85,B 0,C 180,E1 -468.169,E2 -468.169} C_VEL
LIN {X 0,Y 608.552,Z 287.235,A -85,B 0,C 180,E1 -470.977,E2 -470.977} C_VEL
LIN {X 0,Y 608.46,Z 274.688,A -85,B 0,C 180,E1 -472.714,E2 -472.714} C_VEL
LIN {X 0,Y 608.442,Z 274.689,A -85,B 0,C 180,E1 -475.3,E2 -475.3} C_VEL
LIN {X 0,Y 608.445,Z 274.69,A -85,B 0,C 180,E1 -477.517,E2 -477.517} C_VEL
LIN {X 0,Y 608.464,Z 274.695,A -85,B 0,C 180,E1 -479.971,E2 -479.971} C_VEL
LIN {X 0,Y 608.453,Z 274.687,A -85,B 0,C 180,E1 -482.879,E2 -482.879} C_VEL
LIN {X 0,Y 608.434,Z 274.689,A -85,B 0,C 180,E1 -485.277,E2 -485.277} C_VEL
LIN {X 0,Y 608.466,Z 274.687,A -85,B 0,C 180,E1 -487.745,E2 -487.745} C_VEL
LIN {X 0,Y 608.446,Z 274.699,A -85,B 0,C 180,E1 -490.328,E2 -490.328} C_VEL
LIN {X 0,Y 608.472,Z 274.684,A -85,B 0,C 180,E1 -493.309,E2 -493.309} C_VEL
LIN {X 0,Y 608.462,Z 274.69,A -85,B 0,C 180,E1 -496.13,E2 -496.13} C_VEL
LIN {X 0,Y 608.448,Z 274.694,A -85,B 0,C 180,E1 -498.823,E2 -498.823} C_VEL
LIN {X 0,Y 608.461,Z 274.686,A -85,B 0,C 180,E1 -501.411,E2 -501.411} C_VEL
LIN {X 0,Y 608.471,Z 274.685,A -85,B 0,C 180,E1 -503.95,E2 -503.95} C_VEL
LIN {X 0,Y 608.462,Z 274.689,A -85,B 0,C 180,E1 -506.329,E2 -506.329} C_VEL
LIN {X 0,Y 608.472,Z 274.693,A -85,B 0,C 180,E1 -508.726,E2 -508.726} C_VEL
LIN {X 0,Y 608.457,Z 274.689,A -85,B 0,C 180,E1 -511.381,E2 -511.381} C_VEL
LIN {X 0,Y 608.439,Z 274.688,A -85,B 0,C 180,E1 -513.964,E2 -513.964} C_VEL
LIN {X 0,Y 608.461,Z 274.685,A -85,B 0,C 180,E1 -516.155,E2 -516.155} C_VEL
LIN {X 0,Y 608.452,Z 274.696,A -85,B 0,C 180,E1 -519.018,E2 -519.018} C_VEL
LIN {X 0,Y 608.436,Z 274.69,A -85,B 0,C 180,E1 -521.828,E2 -521.828} C_VEL
LIN {X 0,Y 608.466,Z 274.686,A -85,B 0,C 180,E1 -524.594,E2 -524.594} C_VEL
LIN {X 0,Y 608.475,Z 274.695,A -85,B 0,C 180,E1 -527.323,E2 -527.323} C_VEL
LIN {X 0,Y 608.437,Z 274.69,A -85,B 0,C 180,E1 -530.022,E2 -530.022} C_VEL
LIN {X 0,Y 608.476,Z 274.684,A -85,B 0,C 180,E1 -532.701,E2 -532.701} C_VEL
LIN {X 0,Y 608.457,Z 274.694,A -85,B 0,C 180,E1 -535.362,E2 -535.362} C_VEL
LIN {X 0,Y 608.435,Z 274.693,A -85,B 0,C 180,E1 -538.014,E2 -538.014} C_VEL
LIN {X 0,Y 608.458,Z 274.686,A -85,B 0,C 180,E1 -540.662,E2 -540.662} C_VEL
LIN {X 0,Y 608.483,Z 274.686,A -85,B 0,C 180,E1 -543.311,E2 -543.311} C_VEL
LIN {X 0,Y 608.461,Z 274.694,A -85,B 0,C 180,E1 -545.967,E2 -545.967} C_VEL
LIN {X 0,Y 608.43,Z 274.69,A -85,B 0,C 180,E1 -548.636,E2 -548.636} C_VEL
LIN {X 0,Y 608.461,Z 274.688,A -85,B 0,C 180,E1 -549.442,E2 -549.442} C_VEL
LIN {X 0,Y 607.78,Z 274.781,A -85,B 0,C 180,E1 -549.995,E2 -549.995} C_VEL
LIN {X 0,Y 604.928,Z 275.139,A -85,B 0,C 180,E1 -550.892,E2 -550.892} C_VEL
LIN {X 0,Y 602.523,Z 275.438,A -85,B 0,C 180,E1 -551.613,E2 -551.613} C_VEL
LIN {X 0,Y 601.485,Z 275.563,A -85,B 0,C 180,E1 -552.17,E2 -552.17} C_VEL
LIN {X 0,Y 601.397,Z 275.57,A -85,B 0,C 180,E1 -552.358,E2 -552.358} C_VEL
LIN {X 0,Y 601.392,Z 275.566,A -85,B 0,C 180,E1 -554.898,E2 -554.898} C_VEL
LIN {X 0,Y 601.398,Z 275.565,A -85,B 0,C 180,E1 -556.987,E2 -556.987} C_VEL
LIN {X 0,Y 601.397,Z 275.57,A -85,B 0,C 180,E1 -559.81,E2 -559.81} C_VEL
LIN {X 0,Y 601.4,Z 275.569,A -85,B 0,C 180,E1 -562.684,E2 -562.684} C_VEL
LIN {X 0,Y 601.383,Z 275.57,A -85,B 0,C 180,E1 -564.88,E2 -564.88} C_VEL
LIN {X 0,Y 601.379,Z 275.568,A -85,B 0,C 180,E1 -567.358,E2 -567.358} C_VEL
LIN {X 0,Y 601.391,Z 275.566,A -85,B 0,C 180,E1 -569.395,E2 -569.395} C_VEL
LIN {X 0,Y 601.392,Z 275.566,A -85,B 0,C 180,E1 -571.728,E2 -571.728} C_VEL
LIN {X 0,Y 601.414,Z 275.567,A -85,B 0,C 180,E1 -574.119,E2 -574.119} C_VEL
LIN {X 0,Y 601.421,Z 275.563,A -85,B 0,C 180,E1 -577.382,E2 -577.382} C_VEL
LIN {X 0,Y 601.388,Z 275.567,A -85,B 0,C 180,E1 -579.997,E2 -579.997} C_VEL
LIN {X 0,Y 601.404,Z 275.573,A -85,B 0,C 180,E1 -582.671,E2 -582.671} C_VEL
LIN {X 0,Y 601.393,Z 275.568,A -85,B 0,C 180,E1 -585.48,E2 -585.48} C_VEL
LIN {X 0,Y 601.414,Z 275.565,A -85,B 0,C 180,E1 -588.408,E2 -588.408} C_VEL
LIN {X 0,Y 601.395,Z 275.569,A -85,B 0,C 180,E1 -591.534,E2 -591.534} C_VEL
LIN {X 0,Y 601.382,Z 275.569,A -85,B 0,C 180,E1 -593.742,E2 -593.742} C_VEL
LIN {X 0,Y 601.398,Z 275.565,A -85,B 0,C 180,E1 -596.07,E2 -596.07} C_VEL
LIN {X 0,Y 601.408,Z 275.565,A -85,B 0,C 180,E1 -598.548,E2 -598.548} C_VEL
LIN {X 0,Y 601.421,Z 275.573,A -85,B 0,C 180,E1 -601.374,E2 -601.374} C_VEL
LIN {X 0,Y 601.381,Z 275.574,A -85,B 0,C 180,E1 -603.636,E2 -603.636} C_VEL
LIN {X 0,Y 601.419,Z 275.566,A -85,B 0,C 180,E1 -605.859,E2 -605.859} C_VEL
LIN {X 0,Y 601.379,Z 275.57,A -85,B 0,C 180,E1 -608.04,E2 -608.04} C_VEL
LIN {X 0,Y 601.371,Z 275.57,A -85,B 0,C 180,E1 -610.19,E2 -610.19} C_VEL
LIN {X 0,Y 601.356,Z 275.571,A -85,B 0,C 180,E1 -612.311,E2 -612.311} C_VEL
LIN {X 0,Y 601.367,Z 275.57,A -85,B 0,C 180,E1 -614.408,E2 -614.408} C_VEL
LIN {X 0,Y 601.39,Z 275.568,A -85,B 0,C 180,E1 -617.172,E2 -617.172} C_VEL
LIN {X 0,Y 601.387,Z 275.576,A -85,B 0,C 180,E1 -619.905,E2 -619.905} C_VEL
LIN {X 0,Y 601.358,Z 275.571,A -85,B 0,C 180,E1 -622.614,E2 -622.614} C_VEL
LIN {X 0,Y 601.372,Z 275.722,A -85,B 0,C 180,E1 -625.266,E2 -625.266} C_VEL
LIN {X 0,Y 601.475,Z 289.499,A -85,B 0,C 180,E1 -627.657,E2 -627.657} C_VEL
LIN {X 0,Y 601.412,Z 305.168,A -85,B 0,C 180,E1 -630.335,E2 -630.335} C_VEL
LIN {X 0,Y 601.386,Z 308.375,A -85,B 0,C 180,E1 -630.879,E2 -630.879} C_VEL
LIN {X 0,Y 601.643,Z 314.17,A -85,B 0,C 180,E1 -630.963,E2 -630.963} C_VEL
LIN {X 0,Y 601.59,Z 415.652,A -85,B 0,C 180,E1 -632.197,E2 -632.197} C_VEL
LIN {X 0,Y 601.545,Z 429.255,A -85,B 0,C 180,E1 -632.512,E2 -632.512} C_VEL
LIN {X 0,Y 601.55,Z 441.478,A -85,B 0,C 180,E1 -632.93,E2 -632.93} C_VEL
LIN {X 0,Y 601.511,Z 452.491,A -85,B 0,C 180,E1 -633.433,E2 -633.433} C_VEL
LIN {X 0,Y 601.502,Z 463.947,A -85,B 0,C 180,E1 -634.104,E2 -634.104} C_VEL
LIN {X 0,Y 601.443,Z 474.299,A -85,B 0,C 180,E1 -634.86,E2 -634.86} C_VEL
LIN {X 0,Y 601.423,Z 481.881,A -85,B 0,C 180,E1 -635.533,E2 -635.533} C_VEL
LIN {X 0,Y 601.417,Z 490.177,A -85,B 0,C 180,E1 -636.401,E2 -636.401} C_VEL
LIN {X 0,Y 601.365,Z 497.845,A -85,B 0,C 180,E1 -637.386,E2 -637.386} C_VEL
LIN {X 0,Y 601.369,Z 504.171,A -85,B 0,C 180,E1 -638.4,E2 -638.4} C_VEL
LIN {X 0,Y 601.347,Z 509.225,A -85,B 0,C 180,E1 -639.417,E2 -639.417} C_VEL
LIN {X 0,Y 601.358,Z 513.143,A -85,B 0,C 180,E1 -640.437,E2 -640.437} C_VEL
LIN {X 0,Y 601.324,Z 516.027,A -85,B 0,C 180,E1 -641.461,E2 -641.461} C_VEL
LIN {X 0,Y 601.342,Z 517.38,A -85,B 0,C 180,E1 -642.144,E2 -642.144} C_VEL
LIN {X 0,Y 601.325,Z 518.33,A -85,B 0,C 180,E1 -642.831,E2 -642.831} C_VEL
LIN {X 0,Y 601.352,Z 518.999,A -85,B 0,C 180,E1 -644.064,E2 -644.064} C_VEL
LIN {X 0,Y 601.315,Z 518.655,A -85,B 0,C 180,E1 -644.9,E2 -644.9} C_VEL
LIN {X 0,Y 601.324,Z 517.938,A -85,B 0,C 180,E1 -645.594,E2 -645.594} C_VEL
LIN {X 0,Y 601.322,Z 516.117,A -85,B 0,C 180,E1 -646.587,E2 -646.587} C_VEL
LIN {X 0,Y 601.326,Z 513.023,A -85,B 0,C 180,E1 -647.691,E2 -647.691} C_VEL
LIN {X 0,Y 601.348,Z 508.682,A -85,B 0,C 180,E1 -648.798,E2 -648.798} C_VEL
LIN {X 0,Y 601.369,Z 502.428,A -85,B 0,C 180,E1 -649.989,E2 -649.989} C_VEL
LIN {X 0,Y 601.374,Z 494.987,A -85,B 0,C 180,E1 -651.095,E2 -651.095} C_VEL
LIN {X 0,Y 601.387,Z 487.788,A -85,B 0,C 180,E1 -651.96,E2 -651.96} C_VEL
LIN {X 0,Y 601.448,Z 477.572,A -85,B 0,C 180,E1 -652.954,E2 -652.954} C_VEL
LIN {X 0,Y 601.462,Z 467.113,A -85,B 0,C 180,E1 -653.774,E2 -653.774} C_VEL
LIN {X 0,Y 601.47,Z 457.153,A -85,B 0,C 180,E1 -654.404,E2 -654.404} C_VEL
LIN {X 0,Y 601.548,Z 444.981,A -85,B 0,C 180,E1 -655.011,E2 -655.011} C_VEL
LIN {X 0,Y 601.525,Z 432.703,A -85,B 0,C 180,E1 -655.474,E2 -655.474} C_VEL
LIN {X 0,Y 601.532,Z 419.675,A -85,B 0,C 180,E1 -655.818,E2 -655.818} C_VEL
LIN {X 0,Y 601.568,Z 404.91,A -85,B 0,C 180,E1 -656.042,E2 -656.042} C_VEL
LIN {X 0,Y 601.513,Z 309.191,A -85,B 0,C 180,E1 -657.19,E2 -657.19} C_VEL
LIN {X 0,Y 601.412,Z 308.414,A -85,B 0,C 180,E1 -657.203,E2 -657.203} C_VEL
LIN {X 0,Y 601.45,Z 292.247,A -85,B 0,C 180,E1 -659.962,E2 -659.962} C_VEL
LIN {X 0,Y 601.492,Z 276.264,A -85,B 0,C 180,E1 -662.725,E2 -662.725} C_VEL
LIN {X 0,Y 601.439,Z 275.563,A -85,B 0,C 180,E1 -662.863,E2 -662.863} C_VEL
LIN {X 0,Y 601.384,Z 275.57,A -85,B 0,C 180,E1 -665.755,E2 -665.755} C_VEL
LIN {X 0,Y 601.429,Z 275.57,A -85,B 0,C 180,E1 -668.47,E2 -668.47} C_VEL
LIN {X 0,Y 601.424,Z 275.562,A -85,B 0,C 180,E1 -671.593,E2 -671.593} C_VEL
LIN {X 0,Y 601.399,Z 275.577,A -85,B 0,C 180,E1 -674.532,E2 -674.532} C_VEL
LIN {X 0,Y 601.415,Z 275.564,A -85,B 0,C 180,E1 -677.409,E2 -677.409} C_VEL
LIN {X 0,Y 601.402,Z 275.566,A -85,B 0,C 180,E1 -680.004,E2 -680.004} C_VEL
LIN {X 0,Y 601.437,Z 275.569,A -85,B 0,C 180,E1 -682.618,E2 -682.618} C_VEL
LIN {X 0,Y 601.427,Z 275.561,A -85,B 0,C 180,E1 -685.881,E2 -685.881} C_VEL
LIN {X 0,Y 601.419,Z 275.567,A -85,B 0,C 180,E1 -688.545,E2 -688.545} C_VEL
LIN {X 0,Y 601.427,Z 275.567,A -85,B 0,C 180,E1 -691.373,E2 -691.373} C_VEL
LIN {X 0,Y 601.4,Z 275.568,A -85,B 0,C 180,E1 -693.636,E2 -693.636} C_VEL
LIN {X 0,Y 601.419,Z 275.564,A -85,B 0,C 180,E1 -696.59,E2 -696.59} C_VEL
LIN {X 0,Y 601.429,Z 275.57,A -85,B 0,C 180,E1 -699.478,E2 -699.478} C_VEL
LIN {X 0,Y 601.39,Z 275.566,A -85,B 0,C 180,E1 -702.311,E2 -702.311} C_VEL
LIN {X 0,Y 601.408,Z 275.564,A -85,B 0,C 180,E1 -704.408,E2 -704.408} C_VEL
LIN {X 0,Y 601.418,Z 275.567,A -85,B 0,C 180,E1 -707.172,E2 -707.172} C_VEL
LIN {X 0,Y 601.426,Z 275.568,A -85,B 0,C 180,E1 -709.905,E2 -709.905} C_VEL
LIN {X 0,Y 601.439,Z 275.56,A -85,B 0,C 180,E1 -712.615,E2 -712.615} C_VEL
LIN {X 0,Y 601.416,Z 275.565,A -85,B 0,C 180,E1 -715.308,E2 -715.308} C_VEL
LIN {X 0,Y 601.427,Z 275.572,A -85,B 0,C 180,E1 -717.991,E2 -717.991} C_VEL
LIN {X 0,Y 601.441,Z 275.56,A -85,B 0,C 180,E1 -720.669,E2 -720.669} C_VEL
LIN {X 0,Y 601.431,Z 275.562,A -85,B 0,C 180,E1 -723.35,E2 -723.35} C_VEL
LIN {X 0,Y 601.404,Z 275.573,A -85,B 0,C 180,E1 -726.037,E2 -726.037} C_VEL
LIN {X 0,Y 601.412,Z 275.566,A -85,B 0,C 180,E1 -728.738,E2 -728.738} C_VEL
LIN {X 0,Y 601.432,Z 275.56,A -85,B 0,C 180,E1 -731.458,E2 -731.458} C_VEL
LIN {X 0,Y 601.419,Z 275.57,A -85,B 0,C 180,E1 -734.205,E2 -734.205} C_VEL
LIN {X 0,Y 601.428,Z 275.564,A -85,B 0,C 180,E1 -736.986,E2 -736.986} C_VEL
LIN {X 0,Y 601.401,Z 275.565,A -85,B 0,C 180,E1 -739.81,E2 -739.81} C_VEL
LIN {X 0,Y 601.415,Z 275.573,A -85,B 0,C 180,E1 -742.606,E2 -742.606} C_VEL
LIN {X 0,Y 601.397,Z 275.574,A -85,B 0,C 180,E1 -744.879,E2 -744.879} C_VEL
LIN {X 0,Y 601.411,Z 275.566,A -85,B 0,C 180,E1 -747.362,E2 -747.362} C_VEL
LIN {X 0,Y 601.428,Z 275.562,A -85,B 0,C 180,E1 -750.164,E2 -750.164} C_VEL
LIN {X 0,Y 601.417,Z 275.569,A -85,B 0,C 180,E1 -752.715,E2 -752.715} C_VEL
LIN {X 0,Y 601.39,Z 275.578,A -85,B 0,C 180,E1 -755.111,E2 -755.111} C_VEL
LIN {X 0,Y 601.436,Z 275.567,A -85,B 0,C 180,E1 -757.419,E2 -757.419} C_VEL
LIN {X 0,Y 601.401,Z 275.565,A -85,B 0,C 180,E1 -759.996,E2 -759.996} C_VEL
LIN {X 0,Y 601.413,Z 275.565,A -85,B 0,C 180,E1 -762.67,E2 -762.67} C_VEL
LIN {X 0,Y 601.399,Z 275.576,A -85,B 0,C 180,E1 -765.48,E2 -765.48} C_VEL
LIN {X 0,Y 601.423,Z 275.562,A -85,B 0,C 180,E1 -768.407,E2 -768.407} C_VEL
LIN {X 0,Y 601.427,Z 275.572,A -85,B 0,C 180,E1 -771.53,E2 -771.53} C_VEL
LIN {X 0,Y 601.384,Z 275.569,A -85,B 0,C 180,E1 -774.245,E2 -774.245} C_VEL
LIN {X 0,Y 601.416,Z 275.563,A -85,B 0,C 180,E1 -776.686,E2 -776.686} C_VEL
LIN {X 0,Y 601.416,Z 275.563,A -85,B 0,C 180,E1 -779.058,E2 -779.058} C_VEL
LIN {X 0,Y 601.43,Z 275.564,A -85,B 0,C 180,E1 -781.373,E2 -781.373} C_VEL
LIN {X 0,Y 601.399,Z 275.57,A -85,B 0,C 180,E1 -783.636,E2 -783.636} C_VEL
LIN {X 0,Y 601.418,Z 275.569,A -85,B 0,C 180,E1 -786.589,E2 -786.589} C_VEL
LIN {X 0,Y 601.421,Z 275.577,A -85,B 0,C 180,E1 -787.136,E2 -787.136} C_VEL
LIN {X 0,Y 601.673,Z 282.05,A -85,B 0,C 180,E1 -788.051,E2 -788.051} C_VEL
LIN {X 0,Y 601.602,Z 302.761,A -85,B 0,C 180,E1 -790.907,E2 -790.907} C_VEL
LIN {X 0,Y 601.525,Z 323.472,A -85,B 0,C 180,E1 -793.715,E2 -793.715} C_VEL
LIN {X 0,Y 601.468,Z 344.183,A -85,B 0,C 180,E1 -796.485,E2 -796.485} C_VEL
LIN {X 0,Y 601.426,Z 346.61,A -85,B 0,C 180,E1 -796.807,E2 -796.807} C_VEL
LIN {X 0,Y 601.667,Z 350.693,A -85,B 0,C 180,E1 -796.876,E2 -796.876} C_VEL
LIN {X 0,Y 601.594,Z 454.929,A -85,B 0,C 180,E1 -798.139,E2 -798.139} C_VEL
LIN {X 0,Y 601.557,Z 468.205,A -85,B 0,C 180,E1 -798.437,E2 -798.437} C_VEL
LIN {X 0,Y 601.542,Z 479.912,A -85,B 0,C 180,E1 -798.826,E2 -798.826} C_VEL
LIN {X 0,Y 601.521,Z 492.627,A -85,B 0,C 180,E1 -799.396,E2 -799.396} C_VEL
LIN {X 0,Y 601.472,Z 504.193,A -85,B 0,C 180,E1 -800.075,E2 -800.075} C_VEL
LIN {X 0,Y 601.444,Z 514.591,A -85,B 0,C 180,E1 -800.839,E2 -800.839} C_VEL
LIN {X 0,Y 601.405,Z 523.012,A -85,B 0,C 180,E1 -801.6,E2 -801.6} C_VEL
LIN {X 0,Y 601.418,Z 530.957,A -85,B 0,C 180,E1 -802.445,E2 -802.445} C_VEL
LIN {X 0,Y 601.366,Z 538.247,A -85,B 0,C 180,E1 -803.401,E2 -803.401} C_VEL
LIN {X 0,Y 601.372,Z 543.864,A -85,B 0,C 180,E1 -804.299,E2 -804.299} C_VEL
LIN {X 0,Y 601.336,Z 548.948,A -85,B 0,C 180,E1 -805.307,E2 -805.307} C_VEL
LIN {X 0,Y 601.367,Z 552.895,A -85,B 0,C 180,E1 -806.314,E2 -806.314} C_VEL
LIN {X 0,Y 601.325,Z 555.808,A -85,B 0,C 180,E1 -807.32,E2 -807.32} C_VEL
LIN {X 0,Y 601.341,Z 557.201,A -85,B 0,C 180,E1 -807.99,E2 -807.99} C_VEL
LIN {X 0,Y 601.339,Z 558.783,A -85,B 0,C 180,E1 -809.33,E2 -809.33} C_VEL
LIN {X 0,Y 601.335,Z 559,A -85,B 0,C 180,E1 -810,E2 -810} C_VEL
LIN {X 0,Y 601.347,Z 558.185,A -85,B 0,C 180,E1 -811.339,E2 -811.339} C_VEL
LIN {X 0,Y 601.341,Z 557.203,A -85,B 0,C 180,E1 -812.009,E2 -812.009} C_VEL
LIN {X 0,Y 601.325,Z 555.811,A -85,B 0,C 180,E1 -812.679,E2 -812.679} C_VEL
LIN {X 0,Y 601.367,Z 552.898,A -85,B 0,C 180,E1 -813.685,E2 -813.685} C_VEL
LIN {X 0,Y 601.336,Z 548.952,A -85,B 0,C 180,E1 -814.692,E2 -814.692} C_VEL
LIN {X 0,Y 601.372,Z 542.88,A -85,B 0,C 180,E1 -815.869,E2 -815.869} C_VEL
LIN {X 0,Y 601.381,Z 536.24,A -85,B 0,C 180,E1 -816.879,E2 -816.879} C_VEL
LIN {X 0,Y 601.4,Z 527.995,A -85,B 0,C 180,E1 -817.892,E2 -817.892} C_VEL
LIN {X 0,Y 601.434,Z 517.606,A -85,B 0,C 180,E1 -818.906,E2 -818.906} C_VEL
LIN {X 0,Y 601.46,Z 506.756,A -85,B 0,C 180,E1 -819.754,E2 -819.754} C_VEL
LIN {X 0,Y 601.494,Z 495.787,A -85,B 0,C 180,E1 -820.434,E2 -820.434} C_VEL
LIN {X 0,Y 601.548,Z 483.685,A -85,B 0,C 180,E1 -821.022,E2 -821.022} C_VEL
LIN {X 0,Y 601.53,Z 471.897,A -85,B 0,C 180,E1 -821.456,E2 -821.456} C_VEL
LIN {X 0,Y 601.576,Z 459.545,A -85,B 0,C 180,E1 -821.775,E2 -821.775} C_VEL
LIN {X 0,Y 601.607,Z 443.787,A -85,B 0,C 180,E1 -822.01,E2 -822.01} C_VEL
LIN {X 0,Y 601.478,Z 347.199,A -85,B 0,C 180,E1 -823.17,E2 -823.17} C_VEL
LIN {X 0,Y 601.455,Z 346.456,A -85,B 0,C 180,E1 -823.213,E2 -823.213} C_VEL
LIN {X 0,Y 601.466,Z 326.068,A -85,B 0,C 180,E1 -825.937,E2 -825.937} C_VEL
LIN {X 0,Y 601.565,Z 306.2,A -85,B 0,C 180,E1 -828.625,E2 -828.625} C_VEL
LIN {X 0,Y 601.653,Z 284.646,A -85,B 0,C 180,E1 -831.589,E2 -831.589} C_VEL
LIN {X 0,Y 601.672,Z 276.879,A -85,B 0,C 180,E1 -832.672,E2 -832.672} C_VEL
LIN {X 0,Y 601.416,Z 275.567,A -85,B 0,C 180,E1 -832.886,E2 -832.886} C_VEL
LIN {X 0,Y 601.398,Z 275.566,A -85,B 0,C 180,E1 -834.878,E2 -834.878} C_VEL
LIN {X 0,Y 601.416,Z 275.572,A -85,B 0,C 180,E1 -837.867,E2 -837.867} C_VEL
LIN {X 0,Y 601.427,Z 275.572,A -85,B 0,C 180,E1 -840.163,E2 -840.163} C_VEL
LIN {X 0,Y 601.418,Z 275.565,A -85,B 0,C 180,E1 -842.714,E2 -842.714} C_VEL
LIN {X 0,Y 601.39,Z 275.566,A -85,B 0,C 180,E1 -845.111,E2 -845.111} C_VEL
LIN {X 0,Y 601.432,Z 275.561,A -85,B 0,C 180,E1 -847.418,E2 -847.418} C_VEL
LIN {X 0,Y 601.397,Z 275.57,A -85,B 0,C 180,E1 -849.995,E2 -849.995} C_VEL
LIN {X 0,Y 601.409,Z 275.571,A -85,B 0,C 180,E1 -852.669,E2 -852.669} C_VEL
LIN {X 0,Y 601.42,Z 275.562,A -85,B 0,C 180,E1 -855.481,E2 -855.481} C_VEL
LIN {X 0,Y 601.422,Z 275.571,A -85,B 0,C 180,E1 -858.406,E2 -858.406} C_VEL
LIN {X 0,Y 601.427,Z 275.569,A -85,B 0,C 180,E1 -860.874,E2 -860.874} C_VEL
LIN {X 0,Y 601.436,Z 275.56,A -85,B 0,C 180,E1 -863.733,E2 -863.733} C_VEL
LIN {X 0,Y 601.423,Z 275.572,A -85,B 0,C 180,E1 -866.686,E2 -866.686} C_VEL
LIN {X 0,Y 601.425,Z 275.569,A -85,B 0,C 180,E1 -869.058,E2 -869.058} C_VEL
LIN {X 0,Y 601.417,Z 275.566,A -85,B 0,C 180,E1 -871.372,E2 -871.372} C_VEL
LIN {X 0,Y 601.397,Z 275.567,A -85,B 0,C 180,E1 -873.636,E2 -873.636} C_VEL
LIN {X 0,Y 601.416,Z 275.566,A -85,B 0,C 180,E1 -876.589,E2 -876.589} C_VEL
LIN {X 0,Y 601.42,Z 275.568,A -85,B 0,C 180,E1 -879.478,E2 -879.478} C_VEL
LIN {X 0,Y 601.388,Z 275.566,A -85,B 0,C 180,E1 -882.311,E2 -882.311} C_VEL
LIN {X 0,Y 601.424,Z 275.57,A -85,B 0,C 180,E1 -885.103,E2 -885.103} C_VEL
LIN {X 0,Y 601.406,Z 275.567,A -85,B 0,C 180,E1 -887.857,E2 -887.857} C_VEL
LIN {X 0,Y 601.415,Z 275.563,A -85,B 0,C 180,E1 -890.584,E2 -890.584} C_VEL
LIN {X 0,Y 601.445,Z 275.568,A -85,B 0,C 180,E1 -893.324,E2 -893.324} C_VEL
LIN {X 0,Y 601.386,Z 275.571,A -85,B 0,C 180,E1 -895.979,E2 -895.979} C_VEL
LIN {X 0,Y 601.406,Z 275.569,A -85,B 0,C 180,E1 -897.991,E2 -897.991} C_VEL
LIN {X 0,Y 601.431,Z 275.561,A -85,B 0,C 180,E1 -900.67,E2 -900.67} C_VEL
LIN {X 0,Y 601.434,Z 275.565,A -85,B 0,C 180,E1 -903.35,E2 -903.35} C_VEL
LIN {X 0,Y 601.409,Z 275.572,A -85,B 0,C 180,E1 -906.037,E2 -906.037} C_VEL
LIN {X 0,Y 601.432,Z 275.569,A -85,B 0,C 180,E1 -908.061,E2 -908.061} C_VEL
LIN {X 0,Y 601.405,Z 275.564,A -85,B 0,C 180,E1 -911.008,E2 -911.008} C_VEL
LIN {X 0,Y 601.397,Z 275.57,A -85,B 0,C 180,E1 -912.358,E2 -912.358} C_VEL
LIN {X 0,Y 600.72,Z 275.652,A -85,B 0,C 180,E1 -912.917,E2 -912.917} C_VEL
LIN {X 0,Y 597.859,Z 276.013,A -85,B 0,C 180,E1 -913.825,E2 -913.825} C_VEL
LIN {X 0,Y 595.451,Z 276.309,A -85,B 0,C 180,E1 -914.555,E2 -914.555} C_VEL
LIN {X 0,Y 594.424,Z 276.434,A -85,B 0,C 180,E1 -915.119,E2 -915.119} C_VEL
LIN {X 0,Y 594.344,Z 276.445,A -85,B 0,C 180,E1 -915.31,E2 -915.31} C_VEL
LIN {X 0,Y 594.367,Z 276.448,A -85,B 0,C 180,E1 -917.905,E2 -917.905} C_VEL
LIN {X 0,Y 594.36,Z 276.443,A -85,B 0,C 180,E1 -920.915,E2 -920.915} C_VEL
LIN {X 0,Y 594.371,Z 276.442,A -85,B 0,C 180,E1 -923.705,E2 -923.705} C_VEL
LIN {X 0,Y 594.352,Z 276.448,A -85,B 0,C 180,E1 -926.701,E2 -926.701} C_VEL
LIN {X 0,Y 594.368,Z 276.443,A -85,B 0,C 180,E1 -928.999,E2 -928.999} C_VEL
LIN {X 0,Y 594.366,Z 276.441,A -85,B 0,C 180,E1 -931.643,E2 -931.643} C_VEL
LIN {X 0,Y 594.366,Z 276.453,A -85,B 0,C 180,E1 -934.581,E2 -934.581} C_VEL
LIN {X 0,Y 594.377,Z 276.44,A -85,B 0,C 180,E1 -937.609,E2 -937.609} C_VEL
LIN {X 0,Y 594.357,Z 276.45,A -85,B 0,C 180,E1 -940.568,E2 -940.568} C_VEL
LIN {X 0,Y 594.343,Z 276.447,A -85,B 0,C 180,E1 -943.302,E2 -943.302} C_VEL
LIN {X 0,Y 594.354,Z 276.443,A -85,B 0,C 180,E1 -946.162,E2 -946.162} C_VEL
LIN {X 0,Y 594.372,Z 276.448,A -85,B 0,C 180,E1 -949.179,E2 -949.179} C_VEL
LIN {X 0,Y 594.363,Z 276.442,A -85,B 0,C 180,E1 -952.059,E2 -952.059} C_VEL
LIN {X 0,Y 594.346,Z 276.447,A -85,B 0,C 180,E1 -954.678,E2 -954.678} C_VEL
LIN {X 0,Y 594.369,Z 276.45,A -85,B 0,C 180,E1 -957.09,E2 -957.09} C_VEL
LIN {X 0,Y 594.344,Z 276.448,A -85,B 0,C 180,E1 -959.679,E2 -959.679} C_VEL
LIN {X 0,Y 594.33,Z 276.449,A -85,B 0,C 180,E1 -961.772,E2 -961.772} C_VEL
LIN {X 0,Y 594.337,Z 276.446,A -85,B 0,C 180,E1 -964.055,E2 -964.055} C_VEL
LIN {X 0,Y 594.346,Z 276.444,A -85,B 0,C 180,E1 -966.295,E2 -966.295} C_VEL
LIN {X 0,Y 594.405,Z 276.442,A -85,B 0,C 180,E1 -969.225,E2 -969.225} C_VEL
LIN {X 0,Y 594.32,Z 276.45,A -85,B 0,C 180,E1 -972.095,E2 -972.095} C_VEL
LIN {X 0,Y 594.33,Z 276.448,A -85,B 0,C 180,E1 -974.219,E2 -974.219} C_VEL
LIN {X 0,Y 594.336,Z 276.447,A -85,B 0,C 180,E1 -976.321,E2 -976.321} C_VEL
LIN {X 0,Y 594.332,Z 276.446,A -85,B 0,C 180,E1 -978.957,E2 -978.957} C_VEL
LIN {X 0,Y 594.35,Z 276.455,A -85,B 0,C 180,E1 -981.843,E2 -981.843} C_VEL
LIN {X 0,Y 594.343,Z 276.448,A -85,B 0,C 180,E1 -984.572,E2 -984.572} C_VEL
LIN {X 0,Y 594.346,Z 276.468,A -85,B 0,C 180,E1 -985.168,E2 -985.168} C_VEL
LIN {X 0,Y 594.422,Z 288.543,A -85,B 0,C 180,E1 -987.29,E2 -987.29} C_VEL
LIN {X 0,Y 594.375,Z 304.185,A -85,B 0,C 180,E1 -990,E2 -990} C_VEL
LIN {X 0,Y 594.332,Z 308.376,A -85,B 0,C 180,E1 -990.72,E2 -990.72} C_VEL
LIN {X 0,Y 594.753,Z 312.115,A -85,B 0,C 180,E1 -990.783,E2 -990.783} C_VEL
LIN {X 0,Y 594.644,Z 415.478,A -85,B 0,C 180,E1 -992.054,E2 -992.054} C_VEL
LIN {X 0,Y 594.579,Z 429.149,A -85,B 0,C 180,E1 -992.371,E2 -992.371} C_VEL
LIN {X 0,Y 594.565,Z 441.407,A -85,B 0,C 180,E1 -992.795,E2 -992.795} C_VEL
LIN {X 0,Y 594.51,Z 452.44,A -85,B 0,C 180,E1 -993.304,E2 -993.304} C_VEL
LIN {X 0,Y 594.472,Z 463.913,A -85,B 0,C 180,E1 -993.983,E2 -993.983} C_VEL
LIN {X 0,Y 594.419,Z 474.265,A -85,B 0,C 180,E1 -994.748,E2 -994.748} C_VEL
LIN {X 0,Y 594.385,Z 481.867,A -85,B 0,C 180,E1 -995.428,E2 -995.428} C_VEL
LIN {X 0,Y 594.363,Z 489.787,A -85,B 0,C 180,E1 -996.265,E2 -996.265} C_VEL
LIN {X 0,Y 594.29,Z 497.827,A -85,B 0,C 180,E1 -997.304,E2 -997.304} C_VEL
LIN {X 0,Y 594.291,Z 503.192,A -85,B 0,C 180,E1 -998.159,E2 -998.159} C_VEL
LIN {X 0,Y 594.264,Z 508.461,A -85,B 0,C 180,E1 -999.187,E2 -999.187} C_VEL
LIN {X 0,Y 594.248,Z 512.561,A -85,B 0,C 180,E1 -1000.219,E2 -1000.219} C_VEL
LIN {X 0,Y 594.251,Z 514.95,A -85,B 0,C 180,E1 -1001.003,E2 -1001.003} C_VEL
LIN {X 0,Y 594.239,Z 517.657,A -85,B 0,C 180,E1 -1002.292,E2 -1002.292} C_VEL
LIN {X 0,Y 594.244,Z 518.517,A -85,B 0,C 180,E1 -1002.986,E2 -1002.986} C_VEL
LIN {X 0,Y 594.264,Z 518.988,A -85,B 0,C 180,E1 -1004.124,E2 -1004.124} C_VEL
LIN {X 0,Y 594.21,Z 518.534,A -85,B 0,C 180,E1 -1005.082,E2 -1005.082} C_VEL
LIN {X 0,Y 594.223,Z 517.678,A -85,B 0,C 180,E1 -1005.785,E2 -1005.785} C_VEL
LIN {X 0,Y 594.238,Z 516.01,A -85,B 0,C 180,E1 -1006.668,E2 -1006.668} C_VEL
LIN {X 0,Y 594.241,Z 512.424,A -85,B 0,C 180,E1 -1007.909,E2 -1007.909} C_VEL
LIN {X 0,Y 594.246,Z 507.629,A -85,B 0,C 180,E1 -1009.078,E2 -1009.078} C_VEL
LIN {X 0,Y 594.298,Z 501.378,A -85,B 0,C 180,E1 -1010.237,E2 -1010.237} C_VEL
LIN {X 0,Y 594.309,Z 495.085,A -85,B 0,C 180,E1 -1011.166,E2 -1011.166} C_VEL
LIN {X 0,Y 594.344,Z 487.816,A -85,B 0,C 180,E1 -1012.052,E2 -1012.052} C_VEL
LIN {X 0,Y 594.41,Z 477.606,A -85,B 0,C 180,E1 -1013.058,E2 -1013.058} C_VEL
LIN {X 0,Y 594.432,Z 467.148,A -85,B 0,C 180,E1 -1013.888,E2 -1013.888} C_VEL
LIN {X 0,Y 594.487,Z 455.974,A -85,B 0,C 180,E1 -1014.593,E2 -1014.593} C_VEL
LIN {X 0,Y 594.554,Z 443.983,A -85,B 0,C 180,E1 -1015.185,E2 -1015.185} C_VEL
LIN {X 0,Y 594.582,Z 431.408,A -85,B 0,C 180,E1 -1015.653,E2 -1015.653} C_VEL
LIN {X 0,Y 594.565,Z 418.883,A -85,B 0,C 180,E1 -1015.974,E2 -1015.974} C_VEL
LIN {X 0,Y 594.628,Z 402.248,A -85,B 0,C 180,E1 -1016.216,E2 -1016.216} C_VEL
LIN {X 0,Y 594.701,Z 310.541,A -85,B 0,C 180,E1 -1017.327,E2 -1017.327} C_VEL
LIN {X 0,Y 594.355,Z 308.39,A -85,B 0,C 180,E1 -1017.367,E2 -1017.367} C_VEL
LIN {X 0,Y 594.445,Z 292.823,A -85,B 0,C 180,E1 -1020.054,E2 -1020.054} C_VEL
LIN {X 0,Y 594.479,Z 277.615,A -85,B 0,C 180,E1 -1022.716,E2 -1022.716} C_VEL
LIN {X 0,Y 594.384,Z 276.443,A -85,B 0,C 180,E1 -1022.95,E2 -1022.95} C_VEL
LIN {X 0,Y 594.349,Z 276.444,A -85,B 0,C 180,E1 -1025.409,E2 -1025.409} C_VEL
LIN {X 0,Y 594.385,Z 276.444,A -85,B 0,C 180,E1 -1027.941,E2 -1027.941} C_VEL
LIN {X 0,Y 594.377,Z 276.444,A -85,B 0,C 180,E1 -1030.822,E2 -1030.822} C_VEL
LIN {X 0,Y 594.368,Z 276.442,A -85,B 0,C 180,E1 -1033.299,E2 -1033.299} C_VEL
LIN {X 0,Y 594.361,Z 276.446,A -85,B 0,C 180,E1 -1036.161,E2 -1036.161} C_VEL
LIN {X 0,Y 594.38,Z 276.449,A -85,B 0,C 180,E1 -1038.536,E2 -1038.536} C_VEL
LIN {X 0,Y 594.382,Z 276.441,A -85,B 0,C 180,E1 -1041.296,E2 -1041.296} C_VEL
LIN {X 0,Y 594.351,Z 276.443,A -85,B 0,C 180,E1 -1043.755,E2 -1043.755} C_VEL
LIN {X 0,Y 594.375,Z 276.442,A -85,B 0,C 180,E1 -1046.238,E2 -1046.238} C_VEL
LIN {X 0,Y 594.369,Z 276.446,A -85,B 0,C 180,E1 -1048.649,E2 -1048.649} C_VEL
LIN {X 0,Y 594.382,Z 276.451,A -85,B 0,C 180,E1 -1051.042,E2 -1051.042} C_VEL
LIN {X 0,Y 594.385,Z 276.439,A -85,B 0,C 180,E1 -1053.977,E2 -1053.977} C_VEL
LIN {X 0,Y 594.388,Z 276.438,A -85,B 0,C 180,E1 -1056.296,E2 -1056.296} C_VEL
LIN {X 0,Y 594.403,Z 276.447,A -85,B 0,C 180,E1 -1059.224,E2 -1059.224} C_VEL
LIN {X 0,Y 594.35,Z 276.444,A -85,B 0,C 180,E1 -1062.095,E2 -1062.095} C_VEL
LIN {X 0,Y 594.362,Z 276.442,A -85,B 0,C 180,E1 -1064.219,E2 -1064.219} C_VEL
LIN {X 0,Y 594.38,Z 276.44,A -85,B 0,C 180,E1 -1066.321,E2 -1066.321} C_VEL
LIN {X 0,Y 594.374,Z 276.443,A -85,B 0,C 180,E1 -1069.095,E2 -1069.095} C_VEL
LIN {X 0,Y 594.408,Z 276.445,A -85,B 0,C 180,E1 -1071.843,E2 -1071.843} C_VEL
LIN {X 0,Y 594.392,Z 276.438,A -85,B 0,C 180,E1 -1074.572,E2 -1074.572} C_VEL
LIN {X 0,Y 594.402,Z 276.438,A -85,B 0,C 180,E1 -1077.289,E2 -1077.289} C_VEL
LIN {X 0,Y 594.413,Z 276.446,A -85,B 0,C 180,E1 -1080,E2 -1080} C_VEL
LIN {X 0,Y 594.4,Z 276.438,A -85,B 0,C 180,E1 -1082.711,E2 -1082.711} C_VEL
LIN {X 0,Y 594.393,Z 276.438,A -85,B 0,C 180,E1 -1085.428,E2 -1085.428} C_VEL
LIN {X 0,Y 594.409,Z 276.446,A -85,B 0,C 180,E1 -1088.157,E2 -1088.157} C_VEL
LIN {X 0,Y 594.386,Z 276.438,A -85,B 0,C 180,E1 -1091.073,E2 -1091.073} C_VEL
LIN {X 0,Y 594.379,Z 276.44,A -85,B 0,C 180,E1 -1093.679,E2 -1093.679} C_VEL
LIN {X 0,Y 594.393,Z 276.445,A -85,B 0,C 180,E1 -1096.72,E2 -1096.72} C_VEL
LIN {X 0,Y 594.366,Z 276.442,A -85,B 0,C 180,E1 -1099.335,E2 -1099.335} C_VEL
LIN {X 0,Y 594.362,Z 276.441,A -85,B 0,C 180,E1 -1101.504,E2 -1101.504} C_VEL
LIN {X 0,Y 594.388,Z 276.444,A -85,B 0,C 180,E1 -1104.446,E2 -1104.446} C_VEL
LIN {X 0,Y 594.381,Z 276.448,A -85,B 0,C 180,E1 -1106.7,E2 -1106.7} C_VEL
LIN {X 0,Y 594.38,Z 276.448,A -85,B 0,C 180,E1 -1108.999,E2 -1108.999} C_VEL
LIN {X 0,Y 594.376,Z 276.441,A -85,B 0,C 180,E1 -1111.643,E2 -1111.643} C_VEL
LIN {X 0,Y 594.375,Z 276.443,A -85,B 0,C 180,E1 -1114.58,E2 -1114.58} C_VEL
LIN {X 0,Y 594.39,Z 276.442,A -85,B 0,C 180,E1 -1117.609,E2 -1117.609} C_VEL
LIN {X 0,Y 594.367,Z 276.442,A -85,B 0,C 180,E1 -1120.567,E2 -1120.567} C_VEL
LIN {X 0,Y 594.368,Z 276.452,A -85,B 0,C 180,E1 -1123.3,E2 -1123.3} C_VEL
LIN {X 0,Y 594.361,Z 276.443,A -85,B 0,C 180,E1 -1126.162,E2 -1126.162} C_VEL
LIN {X 0,Y 594.381,Z 276.439,A -85,B 0,C 180,E1 -1128.536,E2 -1128.536} C_VEL
LIN {X 0,Y 594.38,Z 276.445,A -85,B 0,C 180,E1 -1131.296,E2 -1131.296} C_VEL
LIN {X 0,Y 594.351,Z 276.453,A -85,B 0,C 180,E1 -1133.755,E2 -1133.755} C_VEL
LIN {X 0,Y 594.366,Z 276.444,A -85,B 0,C 180,E1 -1136.238,E2 -1136.238} C_VEL
LIN {X 0,Y 594.37,Z 276.441,A -85,B 0,C 180,E1 -1138.65,E2 -1138.65} C_VEL
LIN {X 0,Y 594.384,Z 276.439,A -85,B 0,C 180,E1 -1141.042,E2 -1141.042} C_VEL
LIN {X 0,Y 594.381,Z 276.451,A -85,B 0,C 180,E1 -1143.979,E2 -1143.979} C_VEL
LIN {X 0,Y 594.386,Z 276.445,A -85,B 0,C 180,E1 -1146.665,E2 -1146.665} C_VEL
LIN {X 0,Y 594.403,Z 276.548,A -85,B 0,C 180,E1 -1146.988,E2 -1146.988} C_VEL
LIN {X 0,Y 594.766,Z 281.022,A -85,B 0,C 180,E1 -1147.637,E2 -1147.637} C_VEL
LIN {X 0,Y 594.637,Z 302.761,A -85,B 0,C 180,E1 -1150.674,E2 -1150.674} C_VEL
LIN {X 0,Y 594.554,Z 323.472,A -85,B 0,C 180,E1 -1153.519,E2 -1153.519} C_VEL
LIN {X 0,Y 594.439,Z 345.478,A -85,B 0,C 180,E1 -1156.496,E2 -1156.496} C_VEL
LIN {X 0,Y 594.442,Z 346.61,A -85,B 0,C 180,E1 -1156.649,E2 -1156.649} C_VEL
LIN {X 0,Y 594.776,Z 350.693,A -85,B 0,C 180,E1 -1156.722,E2 -1156.722} C_VEL
LIN {X 0,Y 594.646,Z 454.928,A -85,B 0,C 180,E1 -1157.998,E2 -1157.998} C_VEL
LIN {X 0,Y 594.621,Z 468.206,A -85,B 0,C 180,E1 -1158.3,E2 -1158.3} C_VEL
LIN {X 0,Y 594.574,Z 480.498,A -85,B 0,C 180,E1 -1158.715,E2 -1158.715} C_VEL
LIN {X 0,Y 594.533,Z 492.625,A -85,B 0,C 180,E1 -1159.27,E2 -1159.27} C_VEL
LIN {X 0,Y 594.46,Z 504.195,A -85,B 0,C 180,E1 -1159.957,E2 -1159.957} C_VEL
LIN {X 0,Y 594.413,Z 514.592,A -85,B 0,C 180,E1 -1160.729,E2 -1160.729} C_VEL
LIN {X 0,Y 594.349,Z 523.025,A -85,B 0,C 180,E1 -1161.5,E2 -1161.5} C_VEL
LIN {X 0,Y 594.347,Z 530.957,A -85,B 0,C 180,E1 -1162.355,E2 -1162.355} C_VEL
LIN {X 0,Y 594.281,Z 538.822,A -85,B 0,C 180,E1 -1163.41,E2 -1163.41} C_VEL
LIN {X 0,Y 594.289,Z 545.678,A -85,B 0,C 180,E1 -1164.571,E2 -1164.571} C_VEL
LIN {X 0,Y 594.27,Z 550.37,A -85,B 0,C 180,E1 -1165.591,E2 -1165.591} C_VEL
LIN {X 0,Y 594.267,Z 553.955,A -85,B 0,C 180,E1 -1166.61,E2 -1166.61} C_VEL
LIN {X 0,Y 594.226,Z 555.808,A -85,B 0,C 180,E1 -1167.288,E2 -1167.288} C_VEL
LIN {X 0,Y 594.24,Z 557.2,A -85,B 0,C 180,E1 -1167.966,E2 -1167.966} C_VEL
LIN {X 0,Y 594.239,Z 558.784,A -85,B 0,C 180,E1 -1169.322,E2 -1169.322} C_VEL
LIN {X 0,Y 594.236,Z 559,A -85,B 0,C 180,E1 -1170,E2 -1170} C_VEL
LIN {X 0,Y 594.247,Z 558.185,A -85,B 0,C 180,E1 -1171.355,E2 -1171.355} C_VEL
LIN {X 0,Y 594.24,Z 557.202,A -85,B 0,C 180,E1 -1172.033,E2 -1172.033} C_VEL
LIN {X 0,Y 594.226,Z 555.811,A -85,B 0,C 180,E1 -1172.711,E2 -1172.711} C_VEL
LIN {X 0,Y 594.288,Z 552.898,A -85,B 0,C 180,E1 -1173.729,E2 -1173.729} C_VEL
LIN {X 0,Y 594.241,Z 548.952,A -85,B 0,C 180,E1 -1174.748,E2 -1174.748} C_VEL
LIN {X 0,Y 594.304,Z 542.881,A -85,B 0,C 180,E1 -1175.939,E2 -1175.939} C_VEL
LIN {X 0,Y 594.307,Z 536.24,A -85,B 0,C 180,E1 -1176.961,E2 -1176.961} C_VEL
LIN {X 0,Y 594.359,Z 527.995,A -85,B 0,C 180,E1 -1177.986,E2 -1177.986} C_VEL
LIN {X 0,Y 594.404,Z 517.607,A -85,B 0,C 180,E1 -1179.013,E2 -1179.013} C_VEL
LIN {X 0,Y 594.448,Z 506.756,A -85,B 0,C 180,E1 -1179.87,E2 -1179.87} C_VEL
LIN {X 0,Y 594.505,Z 495.789,A -85,B 0,C 180,E1 -1180.558,E2 -1180.558} C_VEL
LIN {X 0,Y 594.566,Z 483.562,A -85,B 0,C 180,E1 -1181.158,E2 -1181.158} C_VEL
LIN {X 0,Y 594.579,Z 471.895,A -85,B 0,C 180,E1 -1181.591,E2 -1181.591} C_VEL
LIN {X 0,Y 594.633,Z 459.544,A -85,B 0,C 180,E1 -1181.915,E2 -1181.915} C_VEL
LIN {X 0,Y 594.689,Z 443.787,A -85,B 0,C 180,E1 -1182.151,E2 -1182.151} C_VEL
LIN {X 0,Y 594.625,Z 348.205,A -85,B 0,C 180,E1 -1183.312,E2 -1183.312} C_VEL
LIN {X 0,Y 594.423,Z 346.456,A -85,B 0,C 180,E1 -1183.372,E2 -1183.372} C_VEL
LIN {X 0,Y 594.478,Z 327.363,A -85,B 0,C 180,E1 -1185.953,E2 -1185.953} C_VEL
LIN {X 0,Y 594.584,Z 307.946,A -85,B 0,C 180,E1 -1188.61,E2 -1188.61} C_VEL
LIN {X 0,Y 594.707,Z 288.318,A -85,B 0,C 180,E1 -1191.337,E2 -1191.337} C_VEL
LIN {X 0,Y 594.672,Z 277.927,A -85,B 0,C 180,E1 -1192.805,E2 -1192.805} C_VEL
LIN {X 0,Y 594.39,Z 276.445,A -85,B 0,C 180,E1 -1193.057,E2 -1193.057} C_VEL
LIN {X 0,Y 594.371,Z 276.443,A -85,B 0,C 180,E1 -1195.192,E2 -1195.192} C_VEL
LIN {X 0,Y 594.385,Z 276.443,A -85,B 0,C 180,E1 -1197.526,E2 -1197.526} C_VEL
LIN {X 0,Y 594.384,Z 276.446,A -85,B 0,C 180,E1 -1200.327,E2 -1200.327} C_VEL
LIN {X 0,Y 594.374,Z 276.441,A -85,B 0,C 180,E1 -1202.949,E2 -1202.949} C_VEL
LIN {X 0,Y 594.346,Z 276.444,A -85,B 0,C 180,E1 -1205.408,E2 -1205.408} C_VEL
LIN {X 0,Y 594.383,Z 276.444,A -85,B 0,C 180,E1 -1207.94,E2 -1207.94} C_VEL
LIN {X 0,Y 594.375,Z 276.444,A -85,B 0,C 180,E1 -1210.821,E2 -1210.821} C_VEL
LIN {X 0,Y 594.362,Z 276.442,A -85,B 0,C 180,E1 -1213.298,E2 -1213.298} C_VEL
LIN {X 0,Y 594.362,Z 276.447,A -85,B 0,C 180,E1 -1216.16,E2 -1216.16} C_VEL
LIN {X 0,Y 594.378,Z 276.451,A -85,B 0,C 180,E1 -1218.536,E2 -1218.536} C_VEL
LIN {X 0,Y 594.381,Z 276.441,A -85,B 0,C 180,E1 -1221.294,E2 -1221.294} C_VEL
LIN {X 0,Y 594.388,Z 276.438,A -85,B 0,C 180,E1 -1223.758,E2 -1223.758} C_VEL
LIN {X 0,Y 594.374,Z 276.443,A -85,B 0,C 180,E1 -1226.238,E2 -1226.238} C_VEL
LIN {X 0,Y 594.385,Z 276.447,A -85,B 0,C 180,E1 -1228.65,E2 -1228.65} C_VEL
LIN {X 0,Y 594.374,Z 276.449,A -85,B 0,C 180,E1 -1231.042,E2 -1231.042} C_VEL
LIN {X 0,Y 594.382,Z 276.439,A -85,B 0,C 180,E1 -1233.975,E2 -1233.975} C_VEL
LIN {X 0,Y 594.383,Z 276.44,A -85,B 0,C 180,E1 -1236.296,E2 -1236.296} C_VEL
LIN {X 0,Y 594.395,Z 276.447,A -85,B 0,C 180,E1 -1239.224,E2 -1239.224} C_VEL
LIN {X 0,Y 594.345,Z 276.444,A -85,B 0,C 180,E1 -1242.095,E2 -1242.095} C_VEL
LIN {X 0,Y 594.358,Z 276.442,A -85,B 0,C 180,E1 -1244.219,E2 -1244.219} C_VEL
LIN {X 0,Y 594.365,Z 276.447,A -85,B 0,C 180,E1 -1247.017,E2 -1247.017} C_VEL
LIN {X 0,Y 594.38,Z 276.444,A -85,B 0,C 180,E1 -1249.784,E2 -1249.784} C_VEL
LIN {X 0,Y 594.392,Z 276.438,A -85,B 0,C 180,E1 -1252.527,E2 -1252.527} C_VEL
LIN {X 0,Y 594.392,Z 276.444,A -85,B 0,C 180,E1 -1255.252,E2 -1255.252} C_VEL
LIN {X 0,Y 594.378,Z 276.445,A -85,B 0,C 180,E1 -1257.967,E2 -1257.967} C_VEL
LIN {X 0,Y 594.403,Z 276.437,A -85,B 0,C 180,E1 -1260.678,E2 -1260.678} C_VEL
LIN {X 0,Y 594.385,Z 276.443,A -85,B 0,C 180,E1 -1263.389,E2 -1263.389} C_VEL
LIN {X 0,Y 594.357,Z 276.449,A -85,B 0,C 180,E1 -1266.109,E2 -1266.109} C_VEL
LIN {X 0,Y 594.403,Z 276.443,A -85,B 0,C 180,E1 -1268.157,E2 -1268.157} C_VEL
LIN {X 0,Y 594.37,Z 276.441,A -85,B 0,C 180,E1 -1271.07,E2 -1271.07} C_VEL
LIN {X 0,Y 594.373,Z 276.445,A -85,B 0,C 180,E1 -1273.679,E2 -1273.679} C_VEL
LIN {X 0,Y 594.344,Z 276.445,A -85,B 0,C 180,E1 -1275.31,E2 -1275.31} C_VEL
LIN {X 0,Y 593.686,Z 276.534,A -85,B 0,C 180,E1 -1275.876,E2 -1275.876} C_VEL
LIN {X 0,Y 590.837,Z 276.894,A -85,B 0,C 180,E1 -1276.794,E2 -1276.794} C_VEL
LIN {X 0,Y 588.426,Z 277.197,A -85,B 0,C 180,E1 -1277.532,E2 -1277.532} C_VEL
LIN {X 0,Y 587.393,Z 277.321,A -85,B 0,C 180,E1 -1278.102,E2 -1278.102} C_VEL
LIN {X 0,Y 587.31,Z 277.328,A -85,B 0,C 180,E1 -1278.295,E2 -1278.295} C_VEL
LIN {X 0,Y 587.321,Z 277.319,A -85,B 0,C 180,E1 -1281.038,E2 -1281.038} C_VEL
LIN {X 0,Y 587.306,Z 277.321,A -85,B 0,C 180,E1 -1283.26,E2 -1283.26} C_VEL
LIN {X 0,Y 587.32,Z 277.319,A -85,B 0,C 180,E1 -1285.517,E2 -1285.517} C_VEL
LIN {X 0,Y 587.314,Z 277.328,A -85,B 0,C 180,E1 -1288.598,E2 -1288.598} C_VEL
LIN {X 0,Y 587.316,Z 277.323,A -85,B 0,C 180,E1 -1290.968,E2 -1290.968} C_VEL
LIN {X 0,Y 587.319,Z 277.319,A -85,B 0,C 180,E1 -1293.398,E2 -1293.398} C_VEL
LIN {X 0,Y 587.281,Z 277.325,A -85,B 0,C 180,E1 -1295.901,E2 -1295.901} C_VEL
LIN {X 0,Y 587.318,Z 277.326,A -85,B 0,C 180,E1 -1298.481,E2 -1298.481} C_VEL
LIN {X 0,Y 587.322,Z 277.323,A -85,B 0,C 180,E1 -1301.158,E2 -1301.158} C_VEL
LIN {X 0,Y 587.295,Z 277.323,A -85,B 0,C 180,E1 -1304.112,E2 -1304.112} C_VEL
LIN {X 0,Y 587.291,Z 277.333,A -85,B 0,C 180,E1 -1306.993,E2 -1306.993} C_VEL
LIN {X 0,Y 587.299,Z 277.322,A -85,B 0,C 180,E1 -1309.746,E2 -1309.746} C_VEL
LIN {X 0,Y 587.334,Z 277.318,A -85,B 0,C 180,E1 -1312.393,E2 -1312.393} C_VEL
LIN {X 0,Y 587.33,Z 277.321,A -85,B 0,C 180,E1 -1315.655,E2 -1315.655} C_VEL
LIN {X 0,Y 587.329,Z 277.318,A -85,B 0,C 180,E1 -1318.231,E2 -1318.231} C_VEL
LIN {X 0,Y 587.338,Z 277.321,A -85,B 0,C 180,E1 -1320.869,E2 -1320.869} C_VEL
LIN {X 0,Y 587.293,Z 277.326,A -85,B 0,C 180,E1 -1323.833,E2 -1323.833} C_VEL
LIN {X 0,Y 587.299,Z 277.323,A -85,B 0,C 180,E1 -1326.741,E2 -1326.741} C_VEL
LIN {X 0,Y 587.316,Z 277.328,A -85,B 0,C 180,E1 -1329.696,E2 -1329.696} C_VEL
LIN {X 0,Y 587.281,Z 277.33,A -85,B 0,C 180,E1 -1331.873,E2 -1331.873} C_VEL
LIN {X 0,Y 587.292,Z 277.327,A -85,B 0,C 180,E1 -1334.025,E2 -1334.025} C_VEL
LIN {X 0,Y 587.323,Z 277.322,A -85,B 0,C 180,E1 -1336.154,E2 -1336.154} C_VEL
LIN {X 0,Y 587.292,Z 277.323,A -85,B 0,C 180,E1 -1338.962,E2 -1338.962} C_VEL
LIN {X 0,Y 587.315,Z 277.33,A -85,B 0,C 180,E1 -1341.745,E2 -1341.745} C_VEL
LIN {X 0,Y 587.313,Z 277.325,A -85,B 0,C 180,E1 -1344.507,E2 -1344.507} C_VEL
LIN {X 0,Y 587.315,Z 277.456,A -85,B 0,C 180,E1 -1345.11,E2 -1345.11} C_VEL
LIN {X 0,Y 587.416,Z 285.645,A -85,B 0,C 180,E1 -1346.571,E2 -1346.571} C_VEL
LIN {X 0,Y 587.378,Z 301.238,A -85,B 0,C 180,E1 -1349.315,E2 -1349.315} C_VEL
LIN {X 0,Y 587.289,Z 308.376,A -85,B 0,C 180,E1 -1350.558,E2 -1350.558} C_VEL
LIN {X 0,Y 587.849,Z 313.577,A -85,B 0,C 180,E1 -1350.643,E2 -1350.643} C_VEL
LIN {X 0,Y 587.721,Z 415.28,A -85,B 0,C 180,E1 -1351.906,E2 -1351.906} C_VEL
LIN {X 0,Y 587.614,Z 428.301,A -85,B 0,C 180,E1 -1352.207,E2 -1352.207} C_VEL
LIN {X 0,Y 587.584,Z 441.335,A -85,B 0,C 180,E1 -1352.657,E2 -1352.657} C_VEL
LIN {X 0,Y 587.534,Z 452.378,A -85,B 0,C 180,E1 -1353.172,E2 -1353.172} C_VEL
LIN {X 0,Y 587.459,Z 463.873,A -85,B 0,C 180,E1 -1353.859,E2 -1353.859} C_VEL
LIN {X 0,Y 587.381,Z 474.236,A -85,B 0,C 180,E1 -1354.633,E2 -1354.633} C_VEL
LIN {X 0,Y 587.331,Z 483.544,A -85,B 0,C 180,E1 -1355.494,E2 -1355.494} C_VEL
LIN {X 0,Y 587.278,Z 491.892,A -85,B 0,C 180,E1 -1356.425,E2 -1356.425} C_VEL
LIN {X 0,Y 587.232,Z 500.055,A -85,B 0,C 180,E1 -1357.565,E2 -1357.565} C_VEL
LIN {X 0,Y 587.213,Z 505.962,A -85,B 0,C 180,E1 -1358.604,E2 -1358.604} C_VEL
LIN {X 0,Y 587.168,Z 510.636,A -85,B 0,C 180,E1 -1359.647,E2 -1359.647} C_VEL
LIN {X 0,Y 587.184,Z 514.197,A -85,B 0,C 180,E1 -1360.692,E2 -1360.692} C_VEL
LIN {X 0,Y 587.155,Z 516.744,A -85,B 0,C 180,E1 -1361.741,E2 -1361.741} C_VEL
LIN {X 0,Y 587.16,Z 517.918,A -85,B 0,C 180,E1 -1362.442,E2 -1362.442} C_VEL
LIN {X 0,Y 587.146,Z 518.64,A -85,B 0,C 180,E1 -1363.146,E2 -1363.146} C_VEL
LIN {X 0,Y 587.162,Z 518.975,A -85,B 0,C 180,E1 -1364.18,E2 -1364.18} C_VEL
LIN {X 0,Y 587.124,Z 518.353,A -85,B 0,C 180,E1 -1365.269,E2 -1365.269} C_VEL
LIN {X 0,Y 587.137,Z 517.398,A -85,B 0,C 180,E1 -1365.981,E2 -1365.981} C_VEL
LIN {X 0,Y 587.147,Z 515.905,A -85,B 0,C 180,E1 -1366.748,E2 -1366.748} C_VEL
LIN {X 0,Y 587.161,Z 513.045,A -85,B 0,C 180,E1 -1367.772,E2 -1367.772} C_VEL
LIN {X 0,Y 587.172,Z 508.326,A -85,B 0,C 180,E1 -1368.99,E2 -1368.99} C_VEL
LIN {X 0,Y 587.203,Z 502.464,A -85,B 0,C 180,E1 -1370.127,E2 -1370.127} C_VEL
LIN {X 0,Y 587.231,Z 495.278,A -85,B 0,C 180,E1 -1371.225,E2 -1371.225} C_VEL
LIN {X 0,Y 587.293,Z 487.842,A -85,B 0,C 180,E1 -1372.145,E2 -1372.145} C_VEL
LIN {X 0,Y 587.381,Z 477.896,A -85,B 0,C 180,E1 -1373.14,E2 -1373.14} C_VEL
LIN {X 0,Y 587.399,Z 467.181,A -85,B 0,C 180,E1 -1374.004,E2 -1374.004} C_VEL
LIN {X 0,Y 587.499,Z 456.742,A -85,B 0,C 180,E1 -1374.677,E2 -1374.677} C_VEL
LIN {X 0,Y 587.586,Z 445.134,A -85,B 0,C 180,E1 -1375.268,E2 -1375.268} C_VEL
LIN {X 0,Y 587.608,Z 432.916,A -85,B 0,C 180,E1 -1375.742,E2 -1375.742} C_VEL
LIN {X 0,Y 587.635,Z 419.846,A -85,B 0,C 180,E1 -1376.097,E2 -1376.097} C_VEL
LIN {X 0,Y 587.694,Z 404.603,A -85,B 0,C 180,E1 -1376.333,E2 -1376.333} C_VEL
LIN {X 0,Y 587.813,Z 311.461,A -85,B 0,C 180,E1 -1377.474,E2 -1377.474} C_VEL
LIN {X 0,Y 587.308,Z 308.296,A -85,B 0,C 180,E1 -1377.546,E2 -1377.546} C_VEL
LIN {X 0,Y 587.412,Z 293.306,A -85,B 0,C 180,E1 -1380.166,E2 -1380.166} C_VEL
LIN {X 0,Y 587.461,Z 278.229,A -85,B 0,C 180,E1 -1382.837,E2 -1382.837} C_VEL
LIN {X 0,Y 587.342,Z 277.321,A -85,B 0,C 180,E1 -1383.049,E2 -1383.049} C_VEL
LIN {X 0,Y 587.297,Z 277.324,A -85,B 0,C 180,E1 -1385.537,E2 -1385.537} C_VEL
LIN {X 0,Y 587.34,Z 277.32,A -85,B 0,C 180,E1 -1387.838,E2 -1387.838} C_VEL
LIN {X 0,Y 587.312,Z 277.329,A -85,B 0,C 180,E1 -1390.255,E2 -1390.255} C_VEL
LIN {X 0,Y 587.317,Z 277.321,A -85,B 0,C 180,E1 -1393.118,E2 -1393.118} C_VEL
LIN {X 0,Y 587.313,Z 277.323,A -85,B 0,C 180,E1 -1396.048,E2 -1396.048} C_VEL
LIN {X 0,Y 587.336,Z 277.324,A -85,B 0,C 180,E1 -1398.925,E2 -1398.925} C_VEL
LIN {X 0,Y 587.329,Z 277.318,A -85,B 0,C 180,E1 -1401.52,E2 -1401.52} C_VEL
LIN {X 0,Y 587.291,Z 277.324,A -85,B 0,C 180,E1 -1404.1,E2 -1404.1} C_VEL
LIN {X 0,Y 587.333,Z 277.323,A -85,B 0,C 180,E1 -1406.603,E2 -1406.603} C_VEL
LIN {X 0,Y 587.337,Z 277.319,A -85,B 0,C 180,E1 -1409.49,E2 -1409.49} C_VEL
LIN {X 0,Y 587.351,Z 277.316,A -85,B 0,C 180,E1 -1412.307,E2 -1412.307} C_VEL
LIN {X 0,Y 587.333,Z 277.318,A -85,B 0,C 180,E1 -1414.483,E2 -1414.483} C_VEL
LIN {X 0,Y 587.319,Z 277.328,A -85,B 0,C 180,E1 -1417.131,E2 -1417.131} C_VEL
LIN {X 0,Y 587.327,Z 277.322,A -85,B 0,C 180,E1 -1419.695,E2 -1419.695} C_VEL
LIN {X 0,Y 587.306,Z 277.324,A -85,B 0,C 180,E1 -1421.873,E2 -1421.873} C_VEL
LIN {X 0,Y 587.321,Z 277.321,A -85,B 0,C 180,E1 -1424.025,E2 -1424.025} C_VEL
LIN {X 0,Y 587.358,Z 277.315,A -85,B 0,C 180,E1 -1426.154,E2 -1426.154} C_VEL
LIN {X 0,Y 587.34,Z 277.318,A -85,B 0,C 180,E1 -1428.962,E2 -1428.962} C_VEL
LIN {X 0,Y 587.362,Z 277.325,A -85,B 0,C 180,E1 -1431.745,E2 -1431.745} C_VEL
LIN {X 0,Y 587.356,Z 277.315,A -85,B 0,C 180,E1 -1434.507,E2 -1434.507} C_VEL
LIN {X 0,Y 587.369,Z 277.314,A -85,B 0,C 180,E1 -1437.257,E2 -1437.257} C_VEL
LIN {X 0,Y 587.382,Z 277.321,A -85,B 0,C 180,E1 -1440,E2 -1440} C_VEL
LIN {X 0,Y 587.367,Z 277.314,A -85,B 0,C 180,E1 -1442.743,E2 -1442.743} C_VEL
LIN {X 0,Y 587.357,Z 277.315,A -85,B 0,C 180,E1 -1445.493,E2 -1445.493} C_VEL
LIN {X 0,Y 587.362,Z 277.325,A -85,B 0,C 180,E1 -1448.255,E2 -1448.255} C_VEL
LIN {X 0,Y 587.347,Z 277.315,A -85,B 0,C 180,E1 -1451.134,E2 -1451.134} C_VEL
LIN {X 0,Y 587.364,Z 277.322,A -85,B 0,C 180,E1 -1454.26,E2 -1454.26} C_VEL
LIN {X 0,Y 587.347,Z 277.315,A -85,B 0,C 180,E1 -1457.406,E2 -1457.406} C_VEL
LIN {X 0,Y 587.313,Z 277.32,A -85,B 0,C 180,E1 -1459.576,E2 -1459.576} C_VEL
LIN {X 0,Y 587.339,Z 277.324,A -85,B 0,C 180,E1 -1462.514,E2 -1462.514} C_VEL
LIN {X 0,Y 587.35,Z 277.326,A -85,B 0,C 180,E1 -1464.759,E2 -1464.759} C_VEL
LIN {X 0,Y 587.328,Z 277.325,A -85,B 0,C 180,E1 -1467.046,E2 -1467.046} C_VEL
LIN {X 0,Y 587.346,Z 277.318,A -85,B 0,C 180,E1 -1469.38,E2 -1469.38} C_VEL
LIN {X 0,Y 587.342,Z 277.316,A -85,B 0,C 180,E1 -1471.836,E2 -1471.836} C_VEL
LIN {X 0,Y 587.341,Z 277.317,A -85,B 0,C 180,E1 -1474.347,E2 -1474.347} C_VEL
LIN {X 0,Y 587.345,Z 277.319,A -85,B 0,C 180,E1 -1477.608,E2 -1477.608} C_VEL
LIN {X 0,Y 587.311,Z 277.32,A -85,B 0,C 180,E1 -1480.255,E2 -1480.255} C_VEL
LIN {X 0,Y 587.317,Z 277.327,A -85,B 0,C 180,E1 -1483.119,E2 -1483.119} C_VEL
LIN {X 0,Y 587.313,Z 277.322,A -85,B 0,C 180,E1 -1486.049,E2 -1486.049} C_VEL
LIN {X 0,Y 587.337,Z 277.319,A -85,B 0,C 180,E1 -1488.925,E2 -1488.925} C_VEL
LIN {X 0,Y 587.327,Z 277.327,A -85,B 0,C 180,E1 -1491.52,E2 -1491.52} C_VEL
LIN {X 0,Y 587.291,Z 277.327,A -85,B 0,C 180,E1 -1494.1,E2 -1494.1} C_VEL
LIN {X 0,Y 587.329,Z 277.318,A -85,B 0,C 180,E1 -1496.603,E2 -1496.603} C_VEL
LIN {X 0,Y 587.339,Z 277.321,A -85,B 0,C 180,E1 -1499.49,E2 -1499.49} C_VEL
LIN {X 0,Y 587.345,Z 277.322,A -85,B 0,C 180,E1 -1502.309,E2 -1502.309} C_VEL
LIN {X 0,Y 587.351,Z 277.317,A -85,B 0,C 180,E1 -1505.241,E2 -1505.241} C_VEL
LIN {X 0,Y 587.356,Z 277.417,A -85,B 0,C 180,E1 -1506.821,E2 -1506.821} C_VEL
LIN {X 0,Y 587.86,Z 280.914,A -85,B 0,C 180,E1 -1507.344,E2 -1507.344} C_VEL
LIN {X 0,Y 587.698,Z 300.172,A -85,B 0,C 180,E1 -1510.073,E2 -1510.073} C_VEL
LIN {X 0,Y 587.569,Z 319.452,A -85,B 0,C 180,E1 -1512.761,E2 -1512.761} C_VEL
LIN {X 0,Y 587.451,Z 341.885,A -85,B 0,C 180,E1 -1515.843,E2 -1515.843} C_VEL
LIN {X 0,Y 587.392,Z 346.61,A -85,B 0,C 180,E1 -1516.485,E2 -1516.485} C_VEL
LIN {X 0,Y 587.87,Z 350.693,A -85,B 0,C 180,E1 -1516.563,E2 -1516.563} C_VEL
LIN {X 0,Y 587.725,Z 454.928,A -85,B 0,C 180,E1 -1517.855,E2 -1517.855} C_VEL
LIN {X 0,Y 587.672,Z 468.207,A -85,B 0,C 180,E1 -1518.16,E2 -1518.16} C_VEL
LIN {X 0,Y 587.603,Z 480.615,A -85,B 0,C 180,E1 -1518.584,E2 -1518.584} C_VEL
LIN {X 0,Y 587.549,Z 492.624,A -85,B 0,C 180,E1 -1519.141,E2 -1519.141} C_VEL
LIN {X 0,Y 587.443,Z 504.197,A -85,B 0,C 180,E1 -1519.836,E2 -1519.836} C_VEL
LIN {X 0,Y 587.392,Z 514.594,A -85,B 0,C 180,E1 -1520.617,E2 -1520.617} C_VEL
LIN {X 0,Y 587.299,Z 523.039,A -85,B 0,C 180,E1 -1521.397,E2 -1521.397} C_VEL
LIN {X 0,Y 587.274,Z 530.957,A -85,B 0,C 180,E1 -1522.262,E2 -1522.262} C_VEL
LIN {X 0,Y 587.23,Z 537.466,A -85,B 0,C 180,E1 -1523.126,E2 -1523.126} C_VEL
LIN {X 0,Y 587.236,Z 543.864,A -85,B 0,C 180,E1 -1524.161,E2 -1524.161} C_VEL
LIN {X 0,Y 587.147,Z 548.948,A -85,B 0,C 180,E1 -1525.193,E2 -1525.193} C_VEL
LIN {X 0,Y 587.212,Z 552.894,A -85,B 0,C 180,E1 -1526.225,E2 -1526.225} C_VEL
LIN {X 0,Y 587.132,Z 555.807,A -85,B 0,C 180,E1 -1527.255,E2 -1527.255} C_VEL
LIN {X 0,Y 587.139,Z 557.199,A -85,B 0,C 180,E1 -1527.942,E2 -1527.942} C_VEL
LIN {X 0,Y 587.14,Z 558.784,A -85,B 0,C 180,E1 -1529.314,E2 -1529.314} C_VEL
LIN {X 0,Y 587.137,Z 559,A -85,B 0,C 180,E1 -1530,E2 -1530} C_VEL
LIN {X 0,Y 587.147,Z 558.186,A -85,B 0,C 180,E1 -1531.371,E2 -1531.371} C_VEL
LIN {X 0,Y 587.139,Z 557.202,A -85,B 0,C 180,E1 -1532.057,E2 -1532.057} C_VEL
LIN {X 0,Y 587.132,Z 555.811,A -85,B 0,C 180,E1 -1532.744,E2 -1532.744} C_VEL
LIN {X 0,Y 587.212,Z 552.898,A -85,B 0,C 180,E1 -1533.774,E2 -1533.774} C_VEL
LIN {X 0,Y 587.147,Z 548.952,A -85,B 0,C 180,E1 -1534.806,E2 -1534.806} C_VEL
LIN {X 0,Y 587.217,Z 542.881,A -85,B 0,C 180,E1 -1536.011,E2 -1536.011} C_VEL
LIN {X 0,Y 587.244,Z 536.241,A -85,B 0,C 180,E1 -1537.046,E2 -1537.046} C_VEL
LIN {X 0,Y 587.297,Z 527.995,A -85,B 0,C 180,E1 -1538.082,E2 -1538.082} C_VEL
LIN {X 0,Y 587.357,Z 517.608,A -85,B 0,C 180,E1 -1539.122,E2 -1539.122} C_VEL
LIN {X 0,Y 587.444,Z 506.756,A -85,B 0,C 180,E1 -1539.989,E2 -1539.989} C_VEL
LIN {X 0,Y 587.521,Z 495.791,A -85,B 0,C 180,E1 -1540.685,E2 -1540.685} C_VEL
LIN {X 0,Y 587.601,Z 483.799,A -85,B 0,C 180,E1 -1541.282,E2 -1541.282} C_VEL
LIN {X 0,Y 587.636,Z 471.893,A -85,B 0,C 180,E1 -1541.73,E2 -1541.73} C_VEL
LIN {X 0,Y 587.688,Z 459.542,A -85,B 0,C 180,E1 -1542.057,E2 -1542.057} C_VEL
LIN {X 0,Y 587.744,Z 443.787,A -85,B 0,C 180,E1 -1542.297,E2 -1542.297} C_VEL
LIN {X 0,Y 587.719,Z 348.763,A -85,B 0,C 180,E1 -1543.465,E2 -1543.465} C_VEL
LIN {X 0,Y 587.392,Z 346.618,A -85,B 0,C 180,E1 -1543.514,E2 -1543.514} C_VEL
LIN {X 0,Y 587.469,Z 328.657,A -85,B 0,C 180,E1 -1545.97,E2 -1545.97} C_VEL
LIN {X 0,Y 587.608,Z 310.535,A -85,B 0,C 180,E1 -1548.478,E2 -1548.478} C_VEL
LIN {X 0,Y 587.787,Z 291.48,A -85,B 0,C 180,E1 -1551.152,E2 -1551.152} C_VEL
LIN {X 0,Y 587.806,Z 279.777,A -85,B 0,C 180,E1 -1552.821,E2 -1552.821} C_VEL
LIN {X 0,Y 587.334,Z 277.324,A -85,B 0,C 180,E1 -1553.205,E2 -1553.205} C_VEL
LIN {X 0,Y 587.33,Z 277.323,A -85,B 0,C 180,E1 -1555.516,E2 -1555.516} C_VEL
LIN {X 0,Y 587.347,Z 277.324,A -85,B 0,C 180,E1 -1557.817,E2 -1557.817} C_VEL
LIN {X 0,Y 587.335,Z 277.321,A -85,B 0,C 180,E1 -1560.509,E2 -1560.509} C_VEL
LIN {X 0,Y 587.33,Z 277.318,A -85,B 0,C 180,E1 -1563.396,E2 -1563.396} C_VEL
LIN {X 0,Y 587.306,Z 277.326,A -85,B 0,C 180,E1 -1565.898,E2 -1565.898} C_VEL
LIN {X 0,Y 587.325,Z 277.326,A -85,B 0,C 180,E1 -1568.478,E2 -1568.478} C_VEL
LIN {X 0,Y 587.333,Z 277.318,A -85,B 0,C 180,E1 -1571.156,E2 -1571.156} C_VEL
LIN {X 0,Y 587.321,Z 277.324,A -85,B 0,C 180,E1 -1574.113,E2 -1574.113} C_VEL
LIN {X 0,Y 587.31,Z 277.324,A -85,B 0,C 180,E1 -1576.993,E2 -1576.993} C_VEL
LIN {X 0,Y 587.313,Z 277.32,A -85,B 0,C 180,E1 -1579.745,E2 -1579.745} C_VEL
LIN {X 0,Y 587.34,Z 277.322,A -85,B 0,C 180,E1 -1582.392,E2 -1582.392} C_VEL
LIN {X 0,Y 587.32,Z 277.327,A -85,B 0,C 180,E1 -1584.944,E2 -1584.944} C_VEL
LIN {X 0,Y 587.332,Z 277.319,A -85,B 0,C 180,E1 -1587.42,E2 -1587.42} C_VEL
LIN {X 0,Y 587.34,Z 277.317,A -85,B 0,C 180,E1 -1589.83,E2 -1589.83} C_VEL
LIN {X 0,Y 587.332,Z 277.329,A -85,B 0,C 180,E1 -1592.954,E2 -1592.954} C_VEL
LIN {X 0,Y 587.344,Z 277.32,A -85,B 0,C 180,E1 -1595.419,E2 -1595.419} C_VEL
LIN {X 0,Y 587.311,Z 277.32,A -85,B 0,C 180,E1 -1598.225,E2 -1598.225} C_VEL
LIN {X 0,Y 587.342,Z 277.327,A -85,B 0,C 180,E1 -1601.151,E2 -1601.151} C_VEL
LIN {X 0,Y 587.315,Z 277.32,A -85,B 0,C 180,E1 -1604.025,E2 -1604.025} C_VEL
LIN {X 0,Y 587.351,Z 277.315,A -85,B 0,C 180,E1 -1606.154,E2 -1606.154} C_VEL
LIN {X 0,Y 587.338,Z 277.321,A -85,B 0,C 180,E1 -1608.962,E2 -1608.962} C_VEL
LIN {X 0,Y 587.359,Z 277.32,A -85,B 0,C 180,E1 -1611.745,E2 -1611.745} C_VEL
LIN {X 0,Y 587.35,Z 277.315,A -85,B 0,C 180,E1 -1614.507,E2 -1614.507} C_VEL
LIN {X 0,Y 587.373,Z 277.317,A -85,B 0,C 180,E1 -1617.257,E2 -1617.257} C_VEL
LIN {X 0,Y 587.367,Z 277.318,A -85,B 0,C 180,E1 -1620,E2 -1620} C_VEL
LIN {X 0,Y 587.357,Z 277.314,A -85,B 0,C 180,E1 -1622.743,E2 -1622.743} C_VEL
LIN {X 0,Y 587.358,Z 277.32,A -85,B 0,C 180,E1 -1625.493,E2 -1625.493} C_VEL
LIN {X 0,Y 587.354,Z 277.319,A -85,B 0,C 180,E1 -1628.255,E2 -1628.255} C_VEL
LIN {X 0,Y 587.337,Z 277.317,A -85,B 0,C 180,E1 -1631.134,E2 -1631.134} C_VEL
LIN {X 0,Y 587.349,Z 277.323,A -85,B 0,C 180,E1 -1633.846,E2 -1633.846} C_VEL
LIN {X 0,Y 587.329,Z 277.319,A -85,B 0,C 180,E1 -1636.812,E2 -1636.812} C_VEL
LIN {X 0,Y 587.31,Z 277.328,A -85,B 0,C 180,E1 -1638.295,E2 -1638.295} C_VEL
LIN {X 0,Y 586.654,Z 277.404,A -85,B 0,C 180,E1 -1638.867,E2 -1638.867} C_VEL
LIN {X 0,Y 583.826,Z 277.758,A -85,B 0,C 180,E1 -1639.796,E2 -1639.796} C_VEL
LIN {X 0,Y 581.421,Z 278.059,A -85,B 0,C 180,E1 -1640.543,E2 -1640.543} C_VEL
LIN {X 0,Y 580.37,Z 278.185,A -85,B 0,C 180,E1 -1641.119,E2 -1641.119} C_VEL
LIN {X 0,Y 580.274,Z 278.197,A -85,B 0,C 180,E1 -1641.314,E2 -1641.314} C_VEL
LIN {X 0,Y 580.289,Z 278.206,A -85,B 0,C 180,E1 -1644.317,E2 -1644.317} C_VEL
LIN {X 0,Y 580.257,Z 278.205,A -85,B 0,C 180,E1 -1646.625,E2 -1646.625} C_VEL
LIN {X 0,Y 580.289,Z 278.195,A -85,B 0,C 180,E1 -1649.31,E2 -1649.31} C_VEL
LIN {X 0,Y 580.29,Z 278.2,A -85,B 0,C 180,E1 -1652.201,E2 -1652.201} C_VEL
LIN {X 0,Y 580.278,Z 278.206,A -85,B 0,C 180,E1 -1654.697,E2 -1654.697} C_VEL
LIN {X 0,Y 580.288,Z 278.197,A -85,B 0,C 180,E1 -1657.269,E2 -1657.269} C_VEL
LIN {X 0,Y 580.279,Z 278.199,A -85,B 0,C 180,E1 -1660.271,E2 -1660.271} C_VEL
LIN {X 0,Y 580.266,Z 278.207,A -85,B 0,C 180,E1 -1662.708,E2 -1662.708} C_VEL
LIN {X 0,Y 580.249,Z 278.201,A -85,B 0,C 180,E1 -1665.612,E2 -1665.612} C_VEL
LIN {X 0,Y 580.268,Z 278.203,A -85,B 0,C 180,E1 -1668.671,E2 -1668.671} C_VEL
LIN {X 0,Y 580.263,Z 278.208,A -85,B 0,C 180,E1 -1670.965,E2 -1670.965} C_VEL
LIN {X 0,Y 580.243,Z 278.203,A -85,B 0,C 180,E1 -1673.596,E2 -1673.596} C_VEL
LIN {X 0,Y 580.27,Z 278.197,A -85,B 0,C 180,E1 -1676.143,E2 -1676.143} C_VEL
LIN {X 0,Y 580.261,Z 278.2,A -85,B 0,C 180,E1 -1678.615,E2 -1678.615} C_VEL
LIN {X 0,Y 580.277,Z 278.202,A -85,B 0,C 180,E1 -1681.024,E2 -1681.024} C_VEL
LIN {X 0,Y 580.25,Z 278.205,A -85,B 0,C 180,E1 -1683.675,E2 -1683.675} C_VEL
LIN {X 0,Y 580.251,Z 278.2,A -85,B 0,C 180,E1 -1686.442,E2 -1686.442} C_VEL
LIN {X 0,Y 580.267,Z 278.207,A -85,B 0,C 180,E1 -1689.438,E2 -1689.438} C_VEL
LIN {X 0,Y 580.242,Z 278.211,A -85,B 0,C 180,E1 -1691.645,E2 -1691.645} C_VEL
LIN {X 0,Y 580.271,Z 278.197,A -85,B 0,C 180,E1 -1694.547,E2 -1694.547} C_VEL
LIN {X 0,Y 580.282,Z 278.201,A -85,B 0,C 180,E1 -1697.409,E2 -1697.409} C_VEL
LIN {X 0,Y 580.22,Z 278.208,A -85,B 0,C 180,E1 -1700.237,E2 -1700.237} C_VEL
LIN {X 0,Y 580.252,Z 278.204,A -85,B 0,C 180,E1 -1702.344,E2 -1702.344} C_VEL
LIN {X 0,Y 580.304,Z 278.2,A -85,B 0,C 180,E1 -1705.007,E2 -1705.007} C_VEL
LIN {X 0,Y 580.41,Z 286.628,A -85,B 0,C 180,E1 -1706.53,E2 -1706.53} C_VEL
LIN {X 0,Y 580.351,Z 302.222,A -85,B 0,C 180,E1 -1709.307,E2 -1709.307} C_VEL
LIN {X 0,Y 580.256,Z 308.375,A -85,B 0,C 180,E1 -1710.391,E2 -1710.391} C_VEL
LIN {X 0,Y 580.951,Z 313.295,A -85,B 0,C 180,E1 -1710.477,E2 -1710.477} C_VEL
LIN {X 0,Y 580.788,Z 415.099,A -85,B 0,C 180,E1 -1711.756,E2 -1711.756} C_VEL
LIN {X 0,Y 580.661,Z 428.19,A -85,B 0,C 180,E1 -1712.06,E2 -1712.06} C_VEL
LIN {X 0,Y 580.629,Z 441.249,A -85,B 0,C 180,E1 -1712.515,E2 -1712.515} C_VEL
LIN {X 0,Y 580.547,Z 452.323,A -85,B 0,C 180,E1 -1713.036,E2 -1713.036} C_VEL
LIN {X 0,Y 580.44,Z 463.834,A -85,B 0,C 180,E1 -1713.732,E2 -1713.732} C_VEL
LIN {X 0,Y 580.346,Z 474.206,A -85,B 0,C 180,E1 -1714.515,E2 -1714.515} C_VEL
LIN {X 0,Y 580.294,Z 483.529,A -85,B 0,C 180,E1 -1715.386,E2 -1715.386} C_VEL
LIN {X 0,Y 580.258,Z 491.322,A -85,B 0,C 180,E1 -1716.258,E2 -1716.258} C_VEL
LIN {X 0,Y 580.142,Z 498.919,A -85,B 0,C 180,E1 -1717.308,E2 -1717.308} C_VEL
LIN {X 0,Y 580.124,Z 505.037,A -85,B 0,C 180,E1 -1718.359,E2 -1718.359} C_VEL
LIN {X 0,Y 580.084,Z 509.905,A -85,B 0,C 180,E1 -1719.414,E2 -1719.414} C_VEL
LIN {X 0,Y 580.093,Z 513.651,A -85,B 0,C 180,E1 -1720.471,E2 -1720.471} C_VEL
LIN {X 0,Y 580.077,Z 515.586,A -85,B 0,C 180,E1 -1721.178,E2 -1721.178} C_VEL
LIN {X 0,Y 580.054,Z 517.079,A -85,B 0,C 180,E1 -1721.887,E2 -1721.887} C_VEL
LIN {X 0,Y 580.05,Z 518.119,A -85,B 0,C 180,E1 -1722.597,E2 -1722.597} C_VEL
LIN {X 0,Y 580.061,Z 518.757,A -85,B 0,C 180,E1 -1723.309,E2 -1723.309} C_VEL
LIN {X 0,Y 580.052,Z 518.964,A -85,B 0,C 180,E1 -1724.235,E2 -1724.235} C_VEL
LIN {X 0,Y 580.02,Z 518.155,A -85,B 0,C 180,E1 -1725.461,E2 -1725.461} C_VEL
LIN {X 0,Y 580.033,Z 517.112,A -85,B 0,C 180,E1 -1726.182,E2 -1726.182} C_VEL
LIN {X 0,Y 580.044,Z 515.601,A -85,B 0,C 180,E1 -1726.906,E2 -1726.906} C_VEL
LIN {X 0,Y 580.081,Z 512.45,A -85,B 0,C 180,E1 -1727.996,E2 -1727.996} C_VEL
LIN {X 0,Y 580.101,Z 508.127,A -85,B 0,C 180,E1 -1729.094,E2 -1729.094} C_VEL
LIN {X 0,Y 580.118,Z 502.481,A -85,B 0,C 180,E1 -1730.199,E2 -1730.199} C_VEL
LIN {X 0,Y 580.179,Z 495.302,A -85,B 0,C 180,E1 -1731.31,E2 -1731.31} C_VEL
LIN {X 0,Y 580.255,Z 487.871,A -85,B 0,C 180,E1 -1732.241,E2 -1732.241} C_VEL
LIN {X 0,Y 580.358,Z 478.344,A -85,B 0,C 180,E1 -1733.211,E2 -1733.211} C_VEL
LIN {X 0,Y 580.377,Z 468.483,A -85,B 0,C 180,E1 -1734.028,E2 -1734.028} C_VEL
LIN {X 0,Y 580.51,Z 457.373,A -85,B 0,C 180,E1 -1734.77,E2 -1734.77} C_VEL
LIN {X 0,Y 580.6,Z 445.205,A -85,B 0,C 180,E1 -1735.402,E2 -1735.402} C_VEL
LIN {X 0,Y 580.654,Z 432.039,A -85,B 0,C 180,E1 -1735.914,E2 -1735.914} C_VEL
LIN {X 0,Y 580.689,Z 419.061,A -85,B 0,C 180,E1 -1736.259,E2 -1736.259} C_VEL
LIN {X 0,Y 580.754,Z 401.958,A -85,B 0,C 180,E1 -1736.515,E2 -1736.515} C_VEL
LIN {X 0,Y 580.857,Z 311.881,A -85,B 0,C 180,E1 -1737.633,E2 -1737.633} C_VEL
LIN {X 0,Y 580.275,Z 308.371,A -85,B 0,C 180,E1 -1737.699,E2 -1737.699} C_VEL
LIN {X 0,Y 580.428,Z 292.173,A -85,B 0,C 180,E1 -1740.567,E2 -1740.567} C_VEL
LIN {X 0,Y 580.464,Z 279.696,A -85,B 0,C 180,E1 -1742.807,E2 -1742.807} C_VEL
LIN {X 0,Y 580.302,Z 278.199,A -85,B 0,C 180,E1 -1743.096,E2 -1743.096} C_VEL
LIN {X 0,Y 580.246,Z 278.205,A -85,B 0,C 180,E1 -1745.756,E2 -1745.756} C_VEL
LIN {X 0,Y 580.289,Z 278.203,A -85,B 0,C 180,E1 -1748.146,E2 -1748.146} C_VEL
LIN {X 0,Y 580.299,Z 278.198,A -85,B 0,C 180,E1 -1750.843,E2 -1750.843} C_VEL
LIN {X 0,Y 580.274,Z 278.198,A -85,B 0,C 180,E1 -1753.658,E2 -1753.658} C_VEL
LIN {X 0,Y 580.276,Z 278.207,A -85,B 0,C 180,E1 -1756.609,E2 -1756.609} C_VEL
LIN {X 0,Y 580.298,Z 278.197,A -85,B 0,C 180,E1 -1759.156,E2 -1759.156} C_VEL
LIN {X 0,Y 580.291,Z 278.195,A -85,B 0,C 180,E1 -1761.927,E2 -1761.927} C_VEL
LIN {X 0,Y 580.251,Z 278.204,A -85,B 0,C 180,E1 -1764.452,E2 -1764.452} C_VEL
LIN {X 0,Y 580.289,Z 278.205,A -85,B 0,C 180,E1 -1766.975,E2 -1766.975} C_VEL
LIN {X 0,Y 580.296,Z 278.197,A -85,B 0,C 180,E1 -1769.425,E2 -1769.425} C_VEL
LIN {X 0,Y 580.297,Z 278.194,A -85,B 0,C 180,E1 -1772.141,E2 -1772.141} C_VEL
LIN {X 0,Y 580.321,Z 278.2,A -85,B 0,C 180,E1 -1775.27,E2 -1775.27} C_VEL
LIN {X 0,Y 580.269,Z 278.198,A -85,B 0,C 180,E1 -1777.947,E2 -1777.947} C_VEL
LIN {X 0,Y 580.299,Z 278.197,A -85,B 0,C 180,E1 -1780.913,E2 -1780.913} C_VEL
LIN {X 0,Y 580.276,Z 278.201,A -85,B 0,C 180,E1 -1783.825,E2 -1783.825} C_VEL
LIN {X 0,Y 580.325,Z 278.193,A -85,B 0,C 180,E1 -1785.983,E2 -1785.983} C_VEL
LIN {X 0,Y 580.304,Z 278.194,A -85,B 0,C 180,E1 -1788.827,E2 -1788.827} C_VEL
LIN {X 0,Y 580.326,Z 278.199,A -85,B 0,C 180,E1 -1791.644,E2 -1791.644} C_VEL
LIN {X 0,Y 580.322,Z 278.192,A -85,B 0,C 180,E1 -1794.44,E2 -1794.44} C_VEL
LIN {X 0,Y 580.336,Z 278.19,A -85,B 0,C 180,E1 -1797.223,E2 -1797.223} C_VEL
LIN {X 0,Y 580.352,Z 278.196,A -85,B 0,C 180,E1 -1800,E2 -1800} C_VEL
LIN {X 0,Y 580.334,Z 278.19,A -85,B 0,C 180,E1 -1802.777,E2 -1802.777} C_VEL
LIN {X 0,Y 580.322,Z 278.192,A -85,B 0,C 180,E1 -1805.56,E2 -1805.56} C_VEL
LIN {X 0,Y 580.326,Z 278.199,A -85,B 0,C 180,E1 -1808.356,E2 -1808.356} C_VEL
LIN {X 0,Y 580.299,Z 278.192,A -85,B 0,C 180,E1 -1811.191,E2 -1811.191} C_VEL
LIN {X 0,Y 580.324,Z 278.195,A -85,B 0,C 180,E1 -1814.017,E2 -1814.017} C_VEL
LIN {X 0,Y 580.312,Z 278.196,A -85,B 0,C 180,E1 -1816.914,E2 -1816.914} C_VEL
LIN {X 0,Y 580.287,Z 278.196,A -85,B 0,C 180,E1 -1819.823,E2 -1819.823} C_VEL
LIN {X 0,Y 580.27,Z 278.198,A -85,B 0,C 180,E1 -1822.053,E2 -1822.053} C_VEL
LIN {X 0,Y 580.305,Z 278.197,A -85,B 0,C 180,E1 -1825.08,E2 -1825.08} C_VEL
LIN {X 0,Y 580.298,Z 278.195,A -85,B 0,C 180,E1 -1828.186,E2 -1828.186} C_VEL
LIN {X 0,Y 580.284,Z 278.201,A -85,B 0,C 180,E1 -1830.695,E2 -1830.695} C_VEL
LIN {X 0,Y 580.282,Z 278.201,A -85,B 0,C 180,E1 -1833.313,E2 -1833.313} C_VEL
LIN {X 0,Y 580.245,Z 278.202,A -85,B 0,C 180,E1 -1835.756,E2 -1835.756} C_VEL
LIN {X 0,Y 580.288,Z 278.195,A -85,B 0,C 180,E1 -1838.146,E2 -1838.146} C_VEL
LIN {X 0,Y 580.298,Z 278.197,A -85,B 0,C 180,E1 -1840.844,E2 -1840.844} C_VEL
LIN {X 0,Y 580.274,Z 278.203,A -85,B 0,C 180,E1 -1843.659,E2 -1843.659} C_VEL
LIN {X 0,Y 580.275,Z 278.197,A -85,B 0,C 180,E1 -1846.61,E2 -1846.61} C_VEL
LIN {X 0,Y 580.299,Z 278.198,A -85,B 0,C 180,E1 -1849.157,E2 -1849.157} C_VEL
LIN {X 0,Y 580.29,Z 278.201,A -85,B 0,C 180,E1 -1851.927,E2 -1851.927} C_VEL
LIN {X 0,Y 580.251,Z 278.201,A -85,B 0,C 180,E1 -1854.453,E2 -1854.453} C_VEL
LIN {X 0,Y 580.29,Z 278.195,A -85,B 0,C 180,E1 -1856.975,E2 -1856.975} C_VEL
LIN {X 0,Y 580.298,Z 278.198,A -85,B 0,C 180,E1 -1859.425,E2 -1859.425} C_VEL
LIN {X 0,Y 580.294,Z 278.203,A -85,B 0,C 180,E1 -1862.143,E2 -1862.143} C_VEL
LIN {X 0,Y 580.323,Z 278.194,A -85,B 0,C 180,E1 -1865.27,E2 -1865.27} C_VEL
LIN {X 0,Y 580.311,Z 278.257,A -85,B 0,C 180,E1 -1866.659,E2 -1866.659} C_VEL
LIN {X 0,Y 580.936,Z 283.344,A -85,B 0,C 180,E1 -1867.412,E2 -1867.412} C_VEL
LIN {X 0,Y 580.752,Z 302.761,A -85,B 0,C 180,E1 -1870.193,E2 -1870.193} C_VEL
LIN {X 0,Y 580.57,Z 322.714,A -85,B 0,C 180,E1 -1873.004,E2 -1873.004} C_VEL
LIN {X 0,Y 580.423,Z 345.478,A -85,B 0,C 180,E1 -1876.164,E2 -1876.164} C_VEL
LIN {X 0,Y 580.398,Z 346.61,A -85,B 0,C 180,E1 -1876.319,E2 -1876.319} C_VEL
LIN {X 0,Y 580.99,Z 352.481,A -85,B 0,C 180,E1 -1876.423,E2 -1876.423} C_VEL
LIN {X 0,Y 580.787,Z 454.928,A -85,B 0,C 180,E1 -1877.707,E2 -1877.707} C_VEL
LIN {X 0,Y 580.73,Z 468.207,A -85,B 0,C 180,E1 -1878.016,E2 -1878.016} C_VEL
LIN {X 0,Y 580.629,Z 480.364,A -85,B 0,C 180,E1 -1878.435,E2 -1878.435} C_VEL
LIN {X 0,Y 580.556,Z 492.622,A -85,B 0,C 180,E1 -1879.008,E2 -1879.008} C_VEL
LIN {X 0,Y 580.421,Z 504.197,A -85,B 0,C 180,E1 -1879.711,E2 -1879.711} C_VEL
LIN {X 0,Y 580.343,Z 514.595,A -85,B 0,C 180,E1 -1880.502,E2 -1880.502} C_VEL
LIN {X 0,Y 580.263,Z 523.052,A -85,B 0,C 180,E1 -1881.292,E2 -1881.292} C_VEL
LIN {X 0,Y 580.222,Z 530.957,A -85,B 0,C 180,E1 -1882.168,E2 -1882.168} C_VEL
LIN {X 0,Y 580.156,Z 538.634,A -85,B 0,C 180,E1 -1883.219,E2 -1883.219} C_VEL
LIN {X 0,Y 580.139,Z 545.678,A -85,B 0,C 180,E1 -1884.438,E2 -1884.438} C_VEL
LIN {X 0,Y 580.108,Z 550.37,A -85,B 0,C 180,E1 -1885.483,E2 -1885.483} C_VEL
LIN {X 0,Y 580.123,Z 553.956,A -85,B 0,C 180,E1 -1886.527,E2 -1886.527} C_VEL
LIN {X 0,Y 580.043,Z 555.807,A -85,B 0,C 180,E1 -1887.222,E2 -1887.222} C_VEL
LIN {X 0,Y 580.038,Z 557.198,A -85,B 0,C 180,E1 -1887.916,E2 -1887.916} C_VEL
LIN {X 0,Y 580.04,Z 558.784,A -85,B 0,C 180,E1 -1889.305,E2 -1889.305} C_VEL
LIN {X 0,Y 580.037,Z 559,A -85,B 0,C 180,E1 -1889.999,E2 -1889.999} C_VEL
LIN {X 0,Y 580.046,Z 558.187,A -85,B 0,C 180,E1 -1891.388,E2 -1891.388} C_VEL
LIN {X 0,Y 580.038,Z 557.201,A -85,B 0,C 180,E1 -1892.083,E2 -1892.083} C_VEL
LIN {X 0,Y 580.043,Z 555.811,A -85,B 0,C 180,E1 -1892.777,E2 -1892.777} C_VEL
LIN {X 0,Y 580.109,Z 552.898,A -85,B 0,C 180,E1 -1893.82,E2 -1893.82} C_VEL
LIN {X 0,Y 580.053,Z 548.951,A -85,B 0,C 180,E1 -1894.865,E2 -1894.865} C_VEL
LIN {X 0,Y 580.14,Z 542.88,A -85,B 0,C 180,E1 -1896.084,E2 -1896.084} C_VEL
LIN {X 0,Y 580.183,Z 536.242,A -85,B 0,C 180,E1 -1897.132,E2 -1897.132} C_VEL
LIN {X 0,Y 580.246,Z 527.996,A -85,B 0,C 180,E1 -1898.181,E2 -1898.181} C_VEL
LIN {X 0,Y 580.332,Z 517.609,A -85,B 0,C 180,E1 -1899.233,E2 -1899.233} C_VEL
LIN {X 0,Y 580.43,Z 507.935,A -85,B 0,C 180,E1 -1900.023,E2 -1900.023} C_VEL
LIN {X 0,Y 580.531,Z 497.338,A -85,B 0,C 180,E1 -1900.726,E2 -1900.726} C_VEL
LIN {X 0,Y 580.612,Z 485.489,A -85,B 0,C 180,E1 -1901.344,E2 -1901.344} C_VEL
LIN {X 0,Y 580.67,Z 473.193,A -85,B 0,C 180,E1 -1901.829,E2 -1901.829} C_VEL
LIN {X 0,Y 580.754,Z 460.548,A -85,B 0,C 180,E1 -1902.181,E2 -1902.181} C_VEL
LIN {X 0,Y 580.834,Z 447.364,A -85,B 0,C 180,E1 -1902.401,E2 -1902.401} C_VEL
LIN {X 0,Y 580.804,Z 349.436,A -85,B 0,C 180,E1 -1903.62,E2 -1903.62} C_VEL
LIN {X 0,Y 580.398,Z 346.618,A -85,B 0,C 180,E1 -1903.68,E2 -1903.68} C_VEL
LIN {X 0,Y 580.544,Z 326.069,A -85,B 0,C 180,E1 -1906.528,E2 -1906.528} C_VEL
LIN {X 0,Y 580.754,Z 305.062,A -85,B 0,C 180,E1 -1909.479,E2 -1909.479} C_VEL
LIN {X 0,Y 580.964,Z 284.646,A -85,B 0,C 180,E1 -1912.398,E2 -1912.398} C_VEL
LIN {X 0,Y 580.634,Z 279.961,A -85,B 0,C 180,E1 -1913.087,E2 -1913.087} C_VEL
LIN {X 0,Y 580.311,Z 278.2,A -85,B 0,C 180,E1 -1913.376,E2 -1913.376} C_VEL
LIN {X 0,Y 580.289,Z 278.205,A -85,B 0,C 180,E1 -1915.848,E2 -1915.848} C_VEL
LIN {X 0,Y 580.299,Z 278.203,A -85,B 0,C 180,E1 -1918.185,E2 -1918.185} C_VEL
LIN {X 0,Y 580.283,Z 278.198,A -85,B 0,C 180,E1 -1920.694,E2 -1920.694} C_VEL
LIN {X 0,Y 580.3,Z 278.194,A -85,B 0,C 180,E1 -1923.315,E2 -1923.315} C_VEL
LIN {X 0,Y 580.265,Z 278.201,A -85,B 0,C 180,E1 -1925.759,E2 -1925.759} C_VEL
LIN {X 0,Y 580.284,Z 278.204,A -85,B 0,C 180,E1 -1928.145,E2 -1928.145} C_VEL
LIN {X 0,Y 580.295,Z 278.197,A -85,B 0,C 180,E1 -1930.842,E2 -1930.842} C_VEL
LIN {X 0,Y 580.274,Z 278.197,A -85,B 0,C 180,E1 -1933.657,E2 -1933.657} C_VEL
LIN {X 0,Y 580.272,Z 278.207,A -85,B 0,C 180,E1 -1936.608,E2 -1936.608} C_VEL
LIN {X 0,Y 580.294,Z 278.196,A -85,B 0,C 180,E1 -1939.156,E2 -1939.156} C_VEL
LIN {X 0,Y 580.285,Z 278.196,A -85,B 0,C 180,E1 -1941.926,E2 -1941.926} C_VEL
LIN {X 0,Y 580.279,Z 278.202,A -85,B 0,C 180,E1 -1944.454,E2 -1944.454} C_VEL
LIN {X 0,Y 580.284,Z 278.203,A -85,B 0,C 180,E1 -1946.975,E2 -1946.975} C_VEL
LIN {X 0,Y 580.303,Z 278.195,A -85,B 0,C 180,E1 -1949.425,E2 -1949.425} C_VEL
LIN {X 0,Y 580.29,Z 278.195,A -85,B 0,C 180,E1 -1952.14,E2 -1952.14} C_VEL
LIN {X 0,Y 580.301,Z 278.203,A -85,B 0,C 180,E1 -1954.92,E2 -1954.92} C_VEL
LIN {X 0,Y 580.262,Z 278.198,A -85,B 0,C 180,E1 -1957.947,E2 -1957.947} C_VEL
LIN {X 0,Y 580.309,Z 278.199,A -85,B 0,C 180,E1 -1960.914,E2 -1960.914} C_VEL
LIN {X 0,Y 580.269,Z 278.199,A -85,B 0,C 180,E1 -1963.825,E2 -1963.825} C_VEL
LIN {X 0,Y 580.317,Z 278.193,A -85,B 0,C 180,E1 -1965.983,E2 -1965.983} C_VEL
LIN {X 0,Y 580.322,Z 278.193,A -85,B 0,C 180,E1 -1968.827,E2 -1968.827} C_VEL
LIN {X 0,Y 580.324,Z 278.198,A -85,B 0,C 180,E1 -1971.644,E2 -1971.644} C_VEL
LIN {X 0,Y 580.315,Z 278.192,A -85,B 0,C 180,E1 -1974.44,E2 -1974.44} C_VEL
LIN {X 0,Y 580.338,Z 278.193,A -85,B 0,C 180,E1 -1977.223,E2 -1977.223} C_VEL
LIN {X 0,Y 580.337,Z 278.194,A -85,B 0,C 180,E1 -1980,E2 -1980} C_VEL
LIN {X 0,Y 580.325,Z 278.19,A -85,B 0,C 180,E1 -1982.777,E2 -1982.777} C_VEL
LIN {X 0,Y 580.321,Z 278.197,A -85,B 0,C 180,E1 -1985.56,E2 -1985.56} C_VEL
LIN {X 0,Y 580.317,Z 278.195,A -85,B 0,C 180,E1 -1988.356,E2 -1988.356} C_VEL
LIN {X 0,Y 580.289,Z 278.195,A -85,B 0,C 180,E1 -1991.191,E2 -1991.191} C_VEL
LIN {X 0,Y 580.306,Z 278.204,A -85,B 0,C 180,E1 -1994.018,E2 -1994.018} C_VEL
LIN {X 0,Y 580.302,Z 278.194,A -85,B 0,C 180,E1 -1996.914,E2 -1996.914} C_VEL
LIN {X 0,Y 580.277,Z 278.201,A -85,B 0,C 180,E1 -1999.823,E2 -1999.823} C_VEL
LIN {X 0,Y 580.274,Z 278.197,A -85,B 0,C 180,E1 -2001.314,E2 -2001.314} C_VEL
LIN {X 0,Y 579.575,Z 278.29,A -85,B 0,C 180,E1 -2001.893,E2 -2001.893} C_VEL
LIN {X 0,Y 576.697,Z 278.645,A -85,B 0,C 180,E1 -2002.833,E2 -2002.833} C_VEL
LIN {X 0,Y 574.303,Z 278.942,A -85,B 0,C 180,E1 -2003.589,E2 -2003.589} C_VEL
LIN {X 0,Y 573.304,Z 279.073,A -85,B 0,C 180,E1 -2004.173,E2 -2004.173} C_VEL
LIN {X 0,Y 573.237,Z 279.077,A -85,B 0,C 180,E1 -2004.371,E2 -2004.371} C_VEL
LIN {X 0,Y 573.194,Z 279.081,A -85,B 0,C 180,E1 -2006.979,E2 -2006.979} C_VEL
LIN {X 0,Y 573.234,Z 279.074,A -85,B 0,C 180,E1 -2009.488,E2 -2009.488} C_VEL
LIN {X 0,Y 573.245,Z 279.082,A -85,B 0,C 180,E1 -2012.646,E2 -2012.646} C_VEL
LIN {X 0,Y 573.196,Z 279.081,A -85,B 0,C 180,E1 -2015.189,E2 -2015.189} C_VEL
LIN {X 0,Y 573.226,Z 279.075,A -85,B 0,C 180,E1 -2017.809,E2 -2017.809} C_VEL
LIN {X 0,Y 573.238,Z 279.08,A -85,B 0,C 180,E1 -2020.526,E2 -2020.526} C_VEL
LIN {X 0,Y 573.202,Z 279.08,A -85,B 0,C 180,E1 -2023.363,E2 -2023.363} C_VEL
LIN {X 0,Y 573.23,Z 279.076,A -85,B 0,C 180,E1 -2026.333,E2 -2026.333} C_VEL
LIN {X 0,Y 573.24,Z 279.076,A -85,B 0,C 180,E1 -2029.476,E2 -2029.476} C_VEL
LIN {X 0,Y 573.222,Z 279.075,A -85,B 0,C 180,E1 -2032.193,E2 -2032.193} C_VEL
LIN {X 0,Y 573.227,Z 279.084,A -85,B 0,C 180,E1 -2035.23,E2 -2035.23} C_VEL
LIN {X 0,Y 573.221,Z 279.075,A -85,B 0,C 180,E1 -2038.184,E2 -2038.184} C_VEL
LIN {X 0,Y 573.229,Z 279.076,A -85,B 0,C 180,E1 -2040.633,E2 -2040.633} C_VEL
LIN {X 0,Y 573.196,Z 279.087,A -85,B 0,C 180,E1 -2043.516,E2 -2043.516} C_VEL
LIN {X 0,Y 573.2,Z 279.079,A -85,B 0,C 180,E1 -2046.134,E2 -2046.134} C_VEL
LIN {X 0,Y 573.251,Z 279.072,A -85,B 0,C 180,E1 -2048.71,E2 -2048.71} C_VEL
LIN {X 0,Y 573.199,Z 279.086,A -85,B 0,C 180,E1 -2051.411,E2 -2051.411} C_VEL
LIN {X 0,Y 573.218,Z 279.087,A -85,B 0,C 180,E1 -2053.622,E2 -2053.622} C_VEL
LIN {X 0,Y 573.239,Z 279.082,A -85,B 0,C 180,E1 -2055.807,E2 -2055.807} C_VEL
LIN {X 0,Y 573.227,Z 279.075,A -85,B 0,C 180,E1 -2058.765,E2 -2058.765} C_VEL
LIN {X 0,Y 573.231,Z 279.081,A -85,B 0,C 180,E1 -2061.54,E2 -2061.54} C_VEL
LIN {X 0,Y 573.254,Z 279.079,A -85,B 0,C 180,E1 -2064.372,E2 -2064.372} C_VEL
LIN {X 0,Y 573.275,Z 279.188,A -85,B 0,C 180,E1 -2064.945,E2 -2064.945} C_VEL
LIN {X 0,Y 573.402,Z 287.611,A -85,B 0,C 180,E1 -2066.487,E2 -2066.487} C_VEL
LIN {X 0,Y 573.325,Z 303.205,A -85,B 0,C 180,E1 -2069.298,E2 -2069.298} C_VEL
LIN {X 0,Y 573.216,Z 308.376,A -85,B 0,C 180,E1 -2070.22,E2 -2070.22} C_VEL
LIN {X 0,Y 574.058,Z 314.751,A -85,B 0,C 180,E1 -2070.329,E2 -2070.329} C_VEL
LIN {X 0,Y 573.868,Z 414.906,A -85,B 0,C 180,E1 -2071.601,E2 -2071.601} C_VEL
LIN {X 0,Y 573.704,Z 428.085,A -85,B 0,C 180,E1 -2071.909,E2 -2071.909} C_VEL
LIN {X 0,Y 573.672,Z 441.165,A -85,B 0,C 180,E1 -2072.37,E2 -2072.37} C_VEL
LIN {X 0,Y 573.583,Z 452.259,A -85,B 0,C 180,E1 -2072.898,E2 -2072.898} C_VEL
LIN {X 0,Y 573.422,Z 463.794,A -85,B 0,C 180,E1 -2073.602,E2 -2073.602} C_VEL
LIN {X 0,Y 573.317,Z 474.175,A -85,B 0,C 180,E1 -2074.395,E2 -2074.395} C_VEL
LIN {X 0,Y 573.24,Z 483.519,A -85,B 0,C 180,E1 -2075.276,E2 -2075.276} C_VEL
LIN {X 0,Y 573.191,Z 491.302,A -85,B 0,C 180,E1 -2076.159,E2 -2076.159} C_VEL
LIN {X 0,Y 573.065,Z 498.902,A -85,B 0,C 180,E1 -2077.222,E2 -2077.222} C_VEL
LIN {X 0,Y 573.053,Z 505.93,A -85,B 0,C 180,E1 -2078.463,E2 -2078.463} C_VEL
LIN {X 0,Y 572.994,Z 510.61,A -85,B 0,C 180,E1 -2079.531,E2 -2079.531} C_VEL
LIN {X 0,Y 573.01,Z 514.177,A -85,B 0,C 180,E1 -2080.602,E2 -2080.602} C_VEL
LIN {X 0,Y 572.979,Z 515.995,A -85,B 0,C 180,E1 -2081.318,E2 -2081.318} C_VEL
LIN {X 0,Y 572.948,Z 517.359,A -85,B 0,C 180,E1 -2082.036,E2 -2082.036} C_VEL
LIN {X 0,Y 572.946,Z 518.316,A -85,B 0,C 180,E1 -2082.756,E2 -2082.756} C_VEL
LIN {X 0,Y 572.97,Z 518.871,A -85,B 0,C 180,E1 -2083.477,E2 -2083.477} C_VEL
LIN {X 0,Y 572.945,Z 518.952,A -85,B 0,C 180,E1 -2084.291,E2 -2084.291} C_VEL
LIN {X 0,Y 572.916,Z 517.95,A -85,B 0,C 180,E1 -2085.657,E2 -2085.657} C_VEL
LIN {X 0,Y 572.945,Z 515.692,A -85,B 0,C 180,E1 -2086.905,E2 -2086.905} C_VEL
LIN {X 0,Y 572.997,Z 511.815,A -85,B 0,C 180,E1 -2088.226,E2 -2088.226} C_VEL
LIN {X 0,Y 573.031,Z 507.293,A -85,B 0,C 180,E1 -2089.339,E2 -2089.339} C_VEL
LIN {X 0,Y 573.065,Z 501.432,A -85,B 0,C 180,E1 -2090.458,E2 -2090.458} C_VEL
LIN {X 0,Y 573.121,Z 493.955,A -85,B 0,C 180,E1 -2091.585,E2 -2091.585} C_VEL
LIN {X 0,Y 573.205,Z 486.196,A -85,B 0,C 180,E1 -2092.529,E2 -2092.529} C_VEL
LIN {X 0,Y 573.307,Z 477.077,A -85,B 0,C 180,E1 -2093.441,E2 -2093.441} C_VEL
LIN {X 0,Y 573.35,Z 467.251,A -85,B 0,C 180,E1 -2094.245,E2 -2094.245} C_VEL
LIN {X 0,Y 573.502,Z 456.951,A -85,B 0,C 180,E1 -2094.928,E2 -2094.928} C_VEL
LIN {X 0,Y 573.65,Z 445.295,A -85,B 0,C 180,E1 -2095.537,E2 -2095.537} C_VEL
LIN {X 0,Y 573.712,Z 433.134,A -85,B 0,C 180,E1 -2096.021,E2 -2096.021} C_VEL
LIN {X 0,Y 573.759,Z 420.071,A -85,B 0,C 180,E1 -2096.388,E2 -2096.388} C_VEL
LIN {X 0,Y 573.852,Z 405.071,A -85,B 0,C 180,E1 -2096.629,E2 -2096.629} C_VEL
LIN {X 0,Y 573.948,Z 312.639,A -85,B 0,C 180,E1 -2097.79,E2 -2097.79} C_VEL
LIN {X 0,Y 573.236,Z 308.337,A -85,B 0,C 180,E1 -2097.876,E2 -2097.876} C_VEL
LIN {X 0,Y 573.409,Z 292.447,A -85,B 0,C 180,E1 -2100.726,E2 -2100.726} C_VEL
LIN {X 0,Y 573.465,Z 280.813,A -85,B 0,C 180,E1 -2102.84,E2 -2102.84} C_VEL
LIN {X 0,Y 573.285,Z 279.073,A -85,B 0,C 180,E1 -2103.166,E2 -2103.166} C_VEL
LIN {X 0,Y 573.217,Z 279.085,A -85,B 0,C 180,E1 -2106.051,E2 -2106.051} C_VEL
LIN {X 0,Y 573.243,Z 279.078,A -85,B 0,C 180,E1 -2108.702,E2 -2108.702} C_VEL
LIN {X 0,Y 573.232,Z 279.075,A -85,B 0,C 180,E1 -2111.593,E2 -2111.593} C_VEL
LIN {X 0,Y 573.224,Z 279.084,A -85,B 0,C 180,E1 -2114.335,E2 -2114.335} C_VEL
LIN {X 0,Y 573.242,Z 279.074,A -85,B 0,C 180,E1 -2117.358,E2 -2117.358} C_VEL
LIN {X 0,Y 573.24,Z 279.079,A -85,B 0,C 180,E1 -2120.392,E2 -2120.392} C_VEL
LIN {X 0,Y 573.253,Z 279.078,A -85,B 0,C 180,E1 -2123.077,E2 -2123.077} C_VEL
LIN {X 0,Y 573.267,Z 279.071,A -85,B 0,C 180,E1 -2125.671,E2 -2125.671} C_VEL
LIN {X 0,Y 573.24,Z 279.074,A -85,B 0,C 180,E1 -2128.184,E2 -2128.184} C_VEL
LIN {X 0,Y 573.264,Z 279.074,A -85,B 0,C 180,E1 -2130.634,E2 -2130.634} C_VEL
LIN {X 0,Y 573.251,Z 279.082,A -85,B 0,C 180,E1 -2133.024,E2 -2133.024} C_VEL
LIN {X 0,Y 573.275,Z 279.076,A -85,B 0,C 180,E1 -2135.366,E2 -2135.366} C_VEL
LIN {X 0,Y 573.228,Z 279.075,A -85,B 0,C 180,E1 -2138.419,E2 -2138.419} C_VEL
LIN {X 0,Y 573.268,Z 279.071,A -85,B 0,C 180,E1 -2140.731,E2 -2140.731} C_VEL
LIN {X 0,Y 573.249,Z 279.079,A -85,B 0,C 180,E1 -2143.622,E2 -2143.622} C_VEL
LIN {X 0,Y 573.272,Z 279.074,A -85,B 0,C 180,E1 -2145.807,E2 -2145.807} C_VEL
LIN {X 0,Y 573.262,Z 279.07,A -85,B 0,C 180,E1 -2148.745,E2 -2148.745} C_VEL
LIN {X 0,Y 573.282,Z 279.074,A -85,B 0,C 180,E1 -2151.54,E2 -2151.54} C_VEL
LIN {X 0,Y 573.288,Z 279.068,A -85,B 0,C 180,E1 -2154.372,E2 -2154.372} C_VEL
LIN {X 0,Y 573.308,Z 279.075,A -85,B 0,C 180,E1 -2157.892,E2 -2157.892} C_VEL
LIN {X 0,Y 573.327,Z 279.061,A -85,B 0,C 180,E1 -2160.702,E2 -2160.702} C_VEL
LIN {X 0,Y 573.302,Z 279.066,A -85,B 0,C 180,E1 -2162.811,E2 -2162.811} C_VEL
LIN {X 0,Y 573.288,Z 279.069,A -85,B 0,C 180,E1 -2165.628,E2 -2165.628} C_VEL
LIN {X 0,Y 573.282,Z 279.074,A -85,B 0,C 180,E1 -2168.46,E2 -2168.46} C_VEL
LIN {X 0,Y 573.271,Z 279.067,A -85,B 0,C 180,E1 -2171.312,E2 -2171.312} C_VEL
LIN {X 0,Y 573.281,Z 279.079,A -85,B 0,C 180,E1 -2174.424,E2 -2174.424} C_VEL
LIN {X 0,Y 573.258,Z 279.072,A -85,B 0,C 180,E1 -2177.112,E2 -2177.112} C_VEL
LIN {X 0,Y 573.242,Z 279.075,A -85,B 0,C 180,E1 -2180.077,E2 -2180.077} C_VEL
LIN {X 0,Y 573.235,Z 279.078,A -85,B 0,C 180,E1 -2182.338,E2 -2182.338} C_VEL
LIN {X 0,Y 573.253,Z 279.072,A -85,B 0,C 180,E1 -2185.41,E2 -2185.41} C_VEL
LIN {X 0,Y 573.251,Z 279.072,A -85,B 0,C 180,E1 -2188.029,E2 -2188.029} C_VEL
LIN {X 0,Y 573.246,Z 279.072,A -85,B 0,C 180,E1 -2190.176,E2 -2190.176} C_VEL
LIN {X 0,Y 573.252,Z 279.076,A -85,B 0,C 180,E1 -2192.645,E2 -2192.645} C_VEL
LIN {X 0,Y 573.206,Z 279.087,A -85,B 0,C 180,E1 -2195.188,E2 -2195.188} C_VEL
LIN {X 0,Y 573.236,Z 279.075,A -85,B 0,C 180,E1 -2197.808,E2 -2197.808} C_VEL
LIN {X 0,Y 573.245,Z 279.073,A -85,B 0,C 180,E1 -2200.525,E2 -2200.525} C_VEL
LIN {X 0,Y 573.238,Z 279.084,A -85,B 0,C 180,E1 -2203.359,E2 -2203.359} C_VEL
LIN {X 0,Y 573.238,Z 279.074,A -85,B 0,C 180,E1 -2206.641,E2 -2206.641} C_VEL
LIN {X 0,Y 573.246,Z 279.083,A -85,B 0,C 180,E1 -2209.475,E2 -2209.475} C_VEL
LIN {X 0,Y 573.236,Z 279.077,A -85,B 0,C 180,E1 -2212.192,E2 -2212.192} C_VEL
LIN {X 0,Y 573.235,Z 279.077,A -85,B 0,C 180,E1 -2215.229,E2 -2215.229} C_VEL
LIN {X 0,Y 573.252,Z 279.082,A -85,B 0,C 180,E1 -2217.772,E2 -2217.772} C_VEL
LIN {X 0,Y 573.266,Z 279.071,A -85,B 0,C 180,E1 -2220.634,E2 -2220.634} C_VEL
LIN {X 0,Y 573.237,Z 279.078,A -85,B 0,C 180,E1 -2223.508,E2 -2223.508} C_VEL
LIN {X 0,Y 573.239,Z 279.085,A -85,B 0,C 180,E1 -2226.135,E2 -2226.135} C_VEL
LIN {X 0,Y 573.289,Z 279.297,A -85,B 0,C 180,E1 -2226.55,E2 -2226.55} C_VEL
LIN {X 0,Y 573.999,Z 284.419,A -85,B 0,C 180,E1 -2227.314,E2 -2227.314} C_VEL
LIN {X 0,Y 573.833,Z 302.761,A -85,B 0,C 180,E1 -2229.944,E2 -2229.944} C_VEL
LIN {X 0,Y 573.587,Z 323.472,A -85,B 0,C 180,E1 -2232.898,E2 -2232.898} C_VEL
LIN {X 0,Y 573.431,Z 344.183,A -85,B 0,C 180,E1 -2235.811,E2 -2235.811} C_VEL
LIN {X 0,Y 573.393,Z 346.61,A -85,B 0,C 180,E1 -2236.149,E2 -2236.149} C_VEL
LIN {X 0,Y 574.112,Z 352.481,A -85,B 0,C 180,E1 -2236.257,E2 -2236.257} C_VEL
LIN {X 0,Y 573.867,Z 454.928,A -85,B 0,C 180,E1 -2237.557,E2 -2237.557} C_VEL
LIN {X 0,Y 573.789,Z 468.207,A -85,B 0,C 180,E1 -2237.869,E2 -2237.869} C_VEL
LIN {X 0,Y 573.676,Z 480.366,A -85,B 0,C 180,E1 -2238.293,E2 -2238.293} C_VEL
LIN {X 0,Y 573.591,Z 492.629,A -85,B 0,C 180,E1 -2238.873,E2 -2238.873} C_VEL
LIN {X 0,Y 573.438,Z 504.195,A -85,B 0,C 180,E1 -2239.585,E2 -2239.585} C_VEL
LIN {X 0,Y 573.329,Z 514.596,A -85,B 0,C 180,E1 -2240.385,E2 -2240.385} C_VEL
LIN {X 0,Y 573.237,Z 523.066,A -85,B 0,C 180,E1 -2241.184,E2 -2241.184} C_VEL
LIN {X 0,Y 573.161,Z 530.957,A -85,B 0,C 180,E1 -2242.071,E2 -2242.071} C_VEL
LIN {X 0,Y 573.075,Z 538.939,A -85,B 0,C 180,E1 -2243.183,E2 -2243.183} C_VEL
LIN {X 0,Y 573.07,Z 545.678,A -85,B 0,C 180,E1 -2244.369,E2 -2244.369} C_VEL
